KUKA KRL program: EPS_2_26115_SA7008_A_20260219035546.src

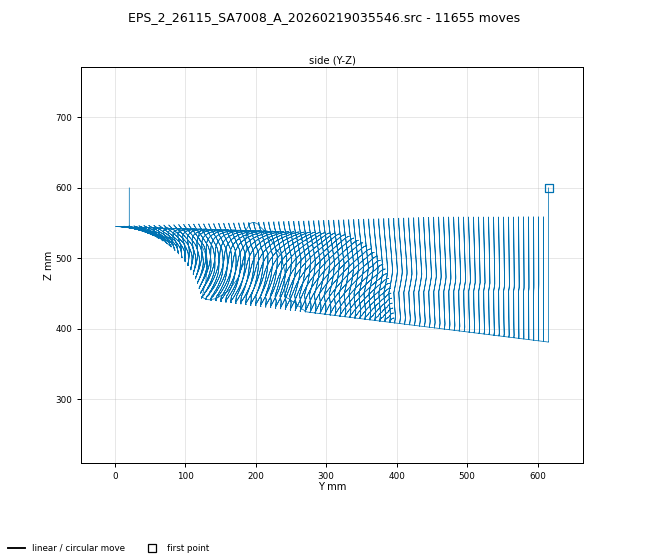
[picture p0: tool path of EPS_2_26115_SA7008_A_20260219035546.src, 11655 of 11657 moves have a stored position in this frame; points joined in program order, loops and branches not executed]
&ACCESS RVP
&REL 4
&COMMENT QRS 19112012
&PARAM EDITMASK = *
DEF PART()
EXT BAS (BAS_COMMAND :IN,REAL :IN )
INT I
BAS (#INITMOV,0 )

;KUKA QRS Post kuka4.cps  Date:22-06-2017 !

File_ID=3064

QRS_PRE_INIT()

;Init var - Until changes are made in qrs_pre_init
Outlet_Square_prg=0
Inlet_1_Square_prg=0
Inlet_2_Square_prg=0
Inlet_3_Square_prg=0
Inlet_4_Square_prg=0
Inlet_5_Square_prg=0

Outlet_1={X 0.000, Y 460.000, Z 458.500, B 0.000, E1 0.000 }
Inlet_1={X 0.000, Y 549.230, Z 433.500, B 0.000, E1 180.000 }
Outlet_1_type=201
Inlet_1_type=0
;QRS#1=Sidecore dimensions
;QRS#2=200-8" PVC SDR 35 Cut Back
;QRS#3=DeadEnd 201
;QRS#4=
;QRS#5=
;QRS#6=
;QRS#7=
;QRS#8=
;QRS#9=12-08 PSX
;QRS#10=

;QRS#11=
;QRS#12=
;QRS#13=
;QRS#14=
;QRS#15=
;QRS#16=1220x127x838 2,75'
;QRS#17=EPS Height
;QRS#18=559
;QRS#19=*
;QRS#20= UPDATED VERSION 22-06-2017
;QRS#21=*
Outlet_Square=0100
Inlet_1_Square=00
Inlet_2_Square=0
Inlet_3_Square=0
Inlet_4_Square=0
Inlet_5_Square=0
Mill_Square=1
Outlet_Square_Prg=214
Inlet_1_Square_prg=0

QRS_INIT()

$ADVANCE=5

; T1
PTP {E1 173.601,E2 173.601}
PTP {X 0,Y 615.5,A -85,B 0,C 180,E1 173.601,E2 173.601,E3 0,E4 0,E5 0,E6 0}
QRS_SPEED_INIT()
LIN {X 0,Y 615.5,Z 600,A -85,B 0,C 180,E1 173.601,E2 173.601,E3 0,E4 0,E5 0,E6 0} C_VEL
LIN {X 0,Y 615.5,Z 391.375,A -85,B 0,C 180,E1 173.601,E2 173.601} C_VEL
LIN {X 0,Y 615.5,Z 383.193,A -85,B 0,C 180,E1 173.601,E2 173.601} C_VEL
LIN {X 0,Y 615.486,Z 381.193,A -85,B 0,C 180,E1 173.415,E2 173.415} C_VEL
LIN {X 0,Y 615.489,Z 381.182,A -85,B 0,C 180,E1 170.802,E2 170.802} C_VEL
LIN {X 0,Y 615.48,Z 381.193,A -85,B 0,C 180,E1 168.139,E2 168.139} C_VEL
LIN {X 0,Y 615.481,Z 381.192,A -85,B 0,C 180,E1 165.451,E2 165.451} C_VEL
LIN {X 0,Y 615.493,Z 381.182,A -85,B 0,C 180,E1 162.73,E2 162.73} C_VEL
LIN {X 0,Y 615.49,Z 381.2,A -85,B 0,C 180,E1 159.968,E2 159.968} C_VEL
LIN {X 0,Y 615.481,Z 381.185,A -85,B 0,C 180,E1 157.156,E2 157.156} C_VEL
LIN {X 0,Y 615.481,Z 381.195,A -85,B 0,C 180,E1 154.284,E2 154.284} C_VEL
LIN {X 0,Y 615.478,Z 381.19,A -85,B 0,C 180,E1 151.55,E2 151.55} C_VEL
LIN {X 0,Y 615.485,Z 381.184,A -85,B 0,C 180,E1 148.913,E2 148.913} C_VEL
LIN {X 0,Y 615.489,Z 381.197,A -85,B 0,C 180,E1 145.979,E2 145.979} C_VEL
LIN {X 0,Y 615.485,Z 381.183,A -85,B 0,C 180,E1 143.062,E2 143.062} C_VEL
LIN {X 0,Y 615.495,Z 381.2,A -85,B 0,C 180,E1 140.251,E2 140.251} C_VEL
LIN {X 0,Y 615.477,Z 381.188,A -85,B 0,C 180,E1 137.647,E2 137.647} C_VEL
LIN {X 0,Y 615.482,Z 381.187,A -85,B 0,C 180,E1 134.932,E2 134.932} C_VEL
LIN {X 0,Y 615.481,Z 381.195,A -85,B 0,C 180,E1 132.08,E2 132.08} C_VEL
LIN {X 0,Y 615.477,Z 381.187,A -85,B 0,C 180,E1 129.75,E2 129.75} C_VEL
LIN {X 0,Y 615.477,Z 381.19,A -85,B 0,C 180,E1 126.936,E2 126.936} C_VEL
LIN {X 0,Y 615.482,Z 381.196,A -85,B 0,C 180,E1 124.701,E2 124.701} C_VEL
LIN {X 0,Y 615.49,Z 381.196,A -85,B 0,C 180,E1 122.332,E2 122.332} C_VEL
LIN {X 0,Y 615.492,Z 381.182,A -85,B 0,C 180,E1 119.405,E2 119.405} C_VEL
LIN {X 0,Y 615.486,Z 381.198,A -85,B 0,C 180,E1 116.444,E2 116.444} C_VEL
LIN {X 0,Y 615.485,Z 381.183,A -85,B 0,C 180,E1 113.556,E2 113.556} C_VEL
LIN {X 0,Y 615.488,Z 381.201,A -85,B 0,C 180,E1 110.73,E2 110.73} C_VEL
LIN {X 0,Y 615.483,Z 381.185,A -85,B 0,C 180,E1 107.957,E2 107.957} C_VEL
LIN {X 0,Y 615.478,Z 381.19,A -85,B 0,C 180,E1 105.226,E2 105.226} C_VEL
LIN {X 0,Y 615.483,Z 381.194,A -85,B 0,C 180,E1 102.53,E2 102.53} C_VEL
LIN {X 0,Y 615.498,Z 381.18,A -85,B 0,C 180,E1 99.862,E2 99.862} C_VEL
LIN {X 0,Y 615.48,Z 381.193,A -85,B 0,C 180,E1 97.215,E2 97.215} C_VEL
LIN {X 0,Y 615.48,Z 381.193,A -85,B 0,C 180,E1 94.584,E2 94.584} C_VEL
LIN {X 0,Y 615.499,Z 381.18,A -85,B 0,C 180,E1 91.963,E2 91.963} C_VEL
LIN {X 0,Y 615.48,Z 381.193,A -85,B 0,C 180,E1 89.346,E2 89.346} C_VEL
LIN {X 0,Y 615.48,Z 381.193,A -85,B 0,C 180,E1 86.727,E2 86.727} C_VEL
LIN {X 0,Y 615.498,Z 381.18,A -85,B 0,C 180,E1 84.101,E2 84.101} C_VEL
LIN {X 0,Y 615.48,Z 381.193,A -85,B 0,C 180,E1 81.463,E2 81.463} C_VEL
LIN {X 0,Y 615.48,Z 381.193,A -85,B 0,C 180,E1 78.807,E2 78.807} C_VEL
LIN {X 0,Y 615.487,Z 381.183,A -85,B 0,C 180,E1 76.065,E2 76.065} C_VEL
LIN {X 0,Y 615.489,Z 381.197,A -85,B 0,C 180,E1 73.414,E2 73.414} C_VEL
LIN {X 0,Y 615.481,Z 381.187,A -85,B 0,C 180,E1 70.662,E2 70.662} C_VEL
LIN {X 0,Y 615.478,Z 381.189,A -85,B 0,C 180,E1 67.863,E2 67.863} C_VEL
LIN {X 0,Y 615.48,Z 381.192,A -85,B 0,C 180,E1 65.008,E2 65.008} C_VEL
LIN {X 0,Y 615.479,Z 381.188,A -85,B 0,C 180,E1 62.823,E2 62.823} C_VEL
LIN {X 0,Y 615.481,Z 381.185,A -85,B 0,C 180,E1 60.205,E2 60.205} C_VEL
LIN {X 0,Y 615.493,Z 381.2,A -85,B 0,C 180,E1 57.543,E2 57.543} C_VEL
LIN {X 0,Y 615.479,Z 381.193,A -85,B 0,C 180,E1 55.185,E2 55.185} C_VEL
LIN {X 0,Y 615.485,Z 381.184,A -85,B 0,C 180,E1 52.758,E2 52.758} C_VEL
LIN {X 0,Y 615.481,Z 381.194,A -85,B 0,C 180,E1 49.911,E2 49.911} C_VEL
LIN {X 0,Y 615.5,Z 381.2,A -85,B 0,C 180,E1 47.649,E2 47.649} C_VEL
LIN {X 0,Y 615.481,Z 381.185,A -85,B 0,C 180,E1 44.932,E2 44.932} C_VEL
LIN {X 0,Y 615.482,Z 381.193,A -85,B 0,C 180,E1 42.08,E2 42.08} C_VEL
LIN {X 0,Y 615.495,Z 381.2,A -85,B 0,C 180,E1 39.749,E2 39.749} C_VEL
LIN {X 0,Y 615.485,Z 381.183,A -85,B 0,C 180,E1 36.937,E2 36.937} C_VEL
LIN {X 0,Y 615.488,Z 381.197,A -85,B 0,C 180,E1 34.021,E2 34.021} C_VEL
LIN {X 0,Y 615.483,Z 381.184,A -85,B 0,C 180,E1 31.086,E2 31.086} C_VEL
LIN {X 0,Y 615.478,Z 381.19,A -85,B 0,C 180,E1 28.45,E2 28.45} C_VEL
LIN {X 0,Y 615.484,Z 381.194,A -85,B 0,C 180,E1 25.715,E2 25.715} C_VEL
LIN {X 0,Y 615.481,Z 381.185,A -85,B 0,C 180,E1 22.844,E2 22.844} C_VEL
LIN {X 0,Y 615.492,Z 381.2,A -85,B 0,C 180,E1 20.032,E2 20.032} C_VEL
LIN {X 0,Y 615.491,Z 381.182,A -85,B 0,C 180,E1 17.27,E2 17.27} C_VEL
LIN {X 0,Y 615.481,Z 381.192,A -85,B 0,C 180,E1 14.549,E2 14.549} C_VEL
LIN {X 0,Y 615.483,Z 381.192,A -85,B 0,C 180,E1 11.86,E2 11.86} C_VEL
LIN {X 0,Y 615.489,Z 381.182,A -85,B 0,C 180,E1 9.198,E2 9.198} C_VEL
LIN {X 0,Y 615.487,Z 381.193,A -85,B 0,C 180,E1 6.556,E2 6.556} C_VEL
LIN {X 0,Y 615.482,Z 381.191,A -85,B 0,C 180,E1 3.928,E2 3.928} C_VEL
LIN {X 0,Y 615.487,Z 381.183,A -85,B 0,C 180,E1 1.308,E2 1.308} C_VEL
LIN {X 0,Y 615.487,Z 381.193,A -85,B 0,C 180,E1 -1.309,E2 -1.309} C_VEL
LIN {X 0,Y 615.483,Z 381.191,A -85,B 0,C 180,E1 -3.929,E2 -3.929} C_VEL
LIN {X 0,Y 615.486,Z 381.183,A -85,B 0,C 180,E1 -6.583,E2 -6.583} C_VEL
LIN {X 0,Y 615.489,Z 381.193,A -85,B 0,C 180,E1 -9.199,E2 -9.199} C_VEL
LIN {X 0,Y 615.483,Z 381.19,A -85,B 0,C 180,E1 -11.861,E2 -11.861} C_VEL
LIN {X 0,Y 615.481,Z 381.184,A -85,B 0,C 180,E1 -14.55,E2 -14.55} C_VEL
LIN {X 0,Y 615.494,Z 381.199,A -85,B 0,C 180,E1 -17.271,E2 -17.271} C_VEL
LIN {X 0,Y 615.491,Z 381.183,A -85,B 0,C 180,E1 -20.033,E2 -20.033} C_VEL
LIN {X 0,Y 615.481,Z 381.191,A -85,B 0,C 180,E1 -22.845,E2 -22.845} C_VEL
LIN {X 0,Y 615.484,Z 381.188,A -85,B 0,C 180,E1 -25.716,E2 -25.716} C_VEL
LIN {X 0,Y 615.478,Z 381.186,A -85,B 0,C 180,E1 -28.45,E2 -28.45} C_VEL
LIN {X 0,Y 615.49,Z 381.201,A -85,B 0,C 180,E1 -31.088,E2 -31.088} C_VEL
LIN {X 0,Y 615.489,Z 381.182,A -85,B 0,C 180,E1 -34.022,E2 -34.022} C_VEL
LIN {X 0,Y 615.493,Z 381.198,A -85,B 0,C 180,E1 -36.938,E2 -36.938} C_VEL
LIN {X 0,Y 615.492,Z 381.183,A -85,B 0,C 180,E1 -39.75,E2 -39.75} C_VEL
LIN {X 0,Y 615.477,Z 381.188,A -85,B 0,C 180,E1 -42.354,E2 -42.354} C_VEL
LIN {X 0,Y 615.491,Z 381.196,A -85,B 0,C 180,E1 -45.069,E2 -45.069} C_VEL
LIN {X 0,Y 615.485,Z 381.183,A -85,B 0,C 180,E1 -47.921,E2 -47.921} C_VEL
LIN {X 0,Y 615.499,Z 381.333,A -85,B 0,C 180,E1 -48.717,E2 -48.717} C_VEL
LIN {X 0,Y 615.485,Z 386.318,A -85,B 0,C 180,E1 -51.096,E2 -51.096} C_VEL
LIN {X 0,Y 615.486,Z 391.692,A -85,B 0,C 180,E1 -53.576,E2 -53.576} C_VEL
LIN {X 0,Y 615.491,Z 398.17,A -85,B 0,C 180,E1 -56.466,E2 -56.466} C_VEL
LIN {X 0,Y 615.478,Z 404.223,A -85,B 0,C 180,E1 -59.08,E2 -59.08} C_VEL
LIN {X 0,Y 615.495,Z 410.088,A -85,B 0,C 180,E1 -61.549,E2 -61.549} C_VEL
LIN {X 0,Y 615.498,Z 417.097,A -85,B 0,C 180,E1 -64.43,E2 -64.43} C_VEL
LIN {X 0,Y 615.483,Z 423.897,A -85,B 0,C 180,E1 -67.155,E2 -67.155} C_VEL
LIN {X 0,Y 615.479,Z 431.039,A -85,B 0,C 180,E1 -69.967,E2 -69.967} C_VEL
LIN {X 0,Y 615.479,Z 438.188,A -85,B 0,C 180,E1 -72.729,E2 -72.729} C_VEL
LIN {X 0,Y 615.483,Z 445.321,A -85,B 0,C 180,E1 -75.451,E2 -75.451} C_VEL
LIN {X 0,Y 615.486,Z 452.468,A -85,B 0,C 180,E1 -78.139,E2 -78.139} C_VEL
LIN {X 0,Y 615.491,Z 453.075,A -85,B 0,C 180,E1 -78.369,E2 -78.369} C_VEL
LIN {X 0,Y 615.493,Z 468.86,A -85,B 0,C 180,E1 -78.724,E2 -78.724} C_VEL
LIN {X 0,Y 615.492,Z 481.787,A -85,B 0,C 180,E1 -79.157,E2 -79.157} C_VEL
LIN {X 0,Y 615.478,Z 494.043,A -85,B 0,C 180,E1 -79.722,E2 -79.722} C_VEL
LIN {X 0,Y 615.498,Z 505.266,A -85,B 0,C 180,E1 -80.387,E2 -80.387} C_VEL
LIN {X 0,Y 615.498,Z 515.389,A -85,B 0,C 180,E1 -81.133,E2 -81.133} C_VEL
LIN {X 0,Y 615.498,Z 524.474,A -85,B 0,C 180,E1 -81.959,E2 -81.959} C_VEL
LIN {X 0,Y 615.498,Z 533.261,A -85,B 0,C 180,E1 -82.943,E2 -82.943} C_VEL
LIN {X 0,Y 615.496,Z 540.416,A -85,B 0,C 180,E1 -83.937,E2 -83.937} C_VEL
LIN {X 0,Y 615.496,Z 546.872,A -85,B 0,C 180,E1 -85.087,E2 -85.087} C_VEL
LIN {X 0,Y 615.496,Z 551.141,A -85,B 0,C 180,E1 -86.071,E2 -86.071} C_VEL
LIN {X 0,Y 615.495,Z 553.398,A -85,B 0,C 180,E1 -86.727,E2 -86.727} C_VEL
LIN {X 0,Y 615.497,Z 555.233,A -85,B 0,C 180,E1 -87.382,E2 -87.382} C_VEL
LIN {X 0,Y 615.499,Z 556.607,A -85,B 0,C 180,E1 -88.037,E2 -88.037} C_VEL
LIN {X 0,Y 615.496,Z 558.173,A -85,B 0,C 180,E1 -89.346,E2 -89.346} C_VEL
LIN {X 0,Y 615.494,Z 558.389,A -85,B 0,C 180,E1 -90,E2 -90} C_VEL
LIN {X 0,Y 615.496,Z 557.58,A -85,B 0,C 180,E1 -91.308,E2 -91.308} C_VEL
LIN {X 0,Y 615.499,Z 556.608,A -85,B 0,C 180,E1 -91.963,E2 -91.963} C_VEL
LIN {X 0,Y 615.497,Z 555.233,A -85,B 0,C 180,E1 -92.618,E2 -92.618} C_VEL
LIN {X 0,Y 615.496,Z 552.35,A -85,B 0,C 180,E1 -93.6,E2 -93.6} C_VEL
LIN {X 0,Y 615.498,Z 548.442,A -85,B 0,C 180,E1 -94.584,E2 -94.584} C_VEL
LIN {X 0,Y 615.499,Z 543.406,A -85,B 0,C 180,E1 -95.569,E2 -95.569} C_VEL
LIN {X 0,Y 615.497,Z 536.87,A -85,B 0,C 180,E1 -96.583,E2 -96.583} C_VEL
LIN {X 0,Y 615.497,Z 529.135,A -85,B 0,C 180,E1 -97.545,E2 -97.545} C_VEL
LIN {X 0,Y 615.498,Z 521.048,A -85,B 0,C 180,E1 -98.371,E2 -98.371} C_VEL
LIN {X 0,Y 615.499,Z 511.171,A -85,B 0,C 180,E1 -99.198,E2 -99.198} C_VEL
LIN {X 0,Y 615.491,Z 499.986,A -85,B 0,C 180,E1 -99.945,E2 -99.945} C_VEL
LIN {X 0,Y 615.481,Z 489.03,A -85,B 0,C 180,E1 -100.527,E2 -100.527} C_VEL
LIN {X 0,Y 615.488,Z 476.477,A -85,B 0,C 180,E1 -101.04,E2 -101.04} C_VEL
LIN {X 0,Y 615.497,Z 464.077,A -85,B 0,C 180,E1 -101.401,E2 -101.401} C_VEL
LIN {X 0,Y 615.491,Z 453.076,A -85,B 0,C 180,E1 -101.631,E2 -101.631} C_VEL
LIN {X 0,Y 615.487,Z 446.962,A -85,B 0,C 180,E1 -103.932,E2 -103.932} C_VEL
LIN {X 0,Y 615.489,Z 439.966,A -85,B 0,C 180,E1 -106.586,E2 -106.586} C_VEL
LIN {X 0,Y 615.481,Z 432.836,A -85,B 0,C 180,E1 -109.338,E2 -109.338} C_VEL
LIN {X 0,Y 615.478,Z 425.679,A -85,B 0,C 180,E1 -112.136,E2 -112.136} C_VEL
LIN {X 0,Y 615.478,Z 418.538,A -85,B 0,C 180,E1 -114.992,E2 -114.992} C_VEL
LIN {X 0,Y 615.478,Z 413.169,A -85,B 0,C 180,E1 -117.177,E2 -117.177} C_VEL
LIN {X 0,Y 615.486,Z 406.877,A -85,B 0,C 180,E1 -119.794,E2 -119.794} C_VEL
LIN {X 0,Y 615.494,Z 400.647,A -85,B 0,C 180,E1 -122.456,E2 -122.456} C_VEL
LIN {X 0,Y 615.479,Z 395.273,A -85,B 0,C 180,E1 -124.815,E2 -124.815} C_VEL
LIN {X 0,Y 615.487,Z 389.901,A -85,B 0,C 180,E1 -127.241,E2 -127.241} C_VEL
LIN {X 0,Y 615.481,Z 383.818,A -85,B 0,C 180,E1 -130.088,E2 -130.088} C_VEL
LIN {X 0,Y 615.494,Z 381.193,A -85,B 0,C 180,E1 -131.378,E2 -131.378} C_VEL
LIN {X 0,Y 615.491,Z 381.182,A -85,B 0,C 180,E1 -134.148,E2 -134.148} C_VEL
LIN {X 0,Y 615.492,Z 381.198,A -85,B 0,C 180,E1 -136.951,E2 -136.951} C_VEL
LIN {X 0,Y 615.481,Z 381.192,A -85,B 0,C 180,E1 -139.393,E2 -139.393} C_VEL
LIN {X 0,Y 615.483,Z 381.183,A -85,B 0,C 180,E1 -141.987,E2 -141.987} C_VEL
LIN {X 0,Y 615.485,Z 381.187,A -85,B 0,C 180,E1 -144.384,E2 -144.384} C_VEL
LIN {X 0,Y 615.484,Z 381.198,A -85,B 0,C 180,E1 -146.763,E2 -146.763} C_VEL
LIN {X 0,Y 615.489,Z 381.195,A -85,B 0,C 180,E1 -149.08,E2 -149.08} C_VEL
LIN {X 0,Y 615.478,Z 381.186,A -85,B 0,C 180,E1 -151.55,E2 -151.55} C_VEL
LIN {X 0,Y 615.484,Z 381.188,A -85,B 0,C 180,E1 -154.284,E2 -154.284} C_VEL
LIN {X 0,Y 615.481,Z 381.191,A -85,B 0,C 180,E1 -157.155,E2 -157.155} C_VEL
LIN {X 0,Y 615.491,Z 381.183,A -85,B 0,C 180,E1 -159.967,E2 -159.967} C_VEL
LIN {X 0,Y 615.494,Z 381.199,A -85,B 0,C 180,E1 -162.729,E2 -162.729} C_VEL
LIN {X 0,Y 615.481,Z 381.184,A -85,B 0,C 180,E1 -165.45,E2 -165.45} C_VEL
LIN {X 0,Y 615.483,Z 381.19,A -85,B 0,C 180,E1 -168.139,E2 -168.139} C_VEL
LIN {X 0,Y 615.489,Z 381.193,A -85,B 0,C 180,E1 -170.801,E2 -170.801} C_VEL
LIN {X 0,Y 615.487,Z 381.182,A -85,B 0,C 180,E1 -173.443,E2 -173.443} C_VEL
LIN {X 0,Y 615.483,Z 381.191,A -85,B 0,C 180,E1 -176.071,E2 -176.071} C_VEL
LIN {X 0,Y 615.487,Z 381.193,A -85,B 0,C 180,E1 -178.691,E2 -178.691} C_VEL
LIN {X 0,Y 615.487,Z 381.183,A -85,B 0,C 180,E1 -181.308,E2 -181.308} C_VEL
LIN {X 0,Y 615.48,Z 381.192,A -85,B 0,C 180,E1 -183.928,E2 -183.928} C_VEL
LIN {X 0,Y 615.486,Z 381.193,A -85,B 0,C 180,E1 -186.585,E2 -186.585} C_VEL
LIN {X 0,Y 614.81,Z 381.332,A -85,B 0,C 180,E1 -187.131,E2 -187.131} C_VEL
LIN {X 0,Y 611.977,Z 381.755,A -85,B 0,C 180,E1 -188.017,E2 -188.017} C_VEL
LIN {X 0,Y 609.586,Z 382.06,A -85,B 0,C 180,E1 -188.729,E2 -188.729} C_VEL
LIN {X 0,Y 608.549,Z 382.177,A -85,B 0,C 180,E1 -189.279,E2 -189.279} C_VEL
LIN {X 0,Y 608.459,Z 382.187,A -85,B 0,C 180,E1 -189.465,E2 -189.465} C_VEL
LIN {X 0,Y 608.456,Z 382.194,A -85,B 0,C 180,E1 -191.999,E2 -191.999} C_VEL
LIN {X 0,Y 608.471,Z 382.187,A -85,B 0,C 180,E1 -194.72,E2 -194.72} C_VEL
LIN {X 0,Y 608.457,Z 382.188,A -85,B 0,C 180,E1 -197.476,E2 -197.476} C_VEL
LIN {X 0,Y 608.46,Z 382.194,A -85,B 0,C 180,E1 -200.274,E2 -200.274} C_VEL
LIN {X 0,Y 608.449,Z 382.191,A -85,B 0,C 180,E1 -202.476,E2 -202.476} C_VEL
LIN {X 0,Y 608.455,Z 382.189,A -85,B 0,C 180,E1 -204.571,E2 -204.571} C_VEL
LIN {X 0,Y 608.483,Z 382.184,A -85,B 0,C 180,E1 -207.21,E2 -207.21} C_VEL
LIN {X 0,Y 608.47,Z 382.195,A -85,B 0,C 180,E1 -209.974,E2 -209.974} C_VEL
LIN {X 0,Y 608.452,Z 382.189,A -85,B 0,C 180,E1 -212.523,E2 -212.523} C_VEL
LIN {X 0,Y 608.442,Z 382.191,A -85,B 0,C 180,E1 -215.277,E2 -215.277} C_VEL
LIN {X 0,Y 608.465,Z 382.196,A -85,B 0,C 180,E1 -217.746,E2 -217.746} C_VEL
LIN {X 0,Y 608.448,Z 382.19,A -85,B 0,C 180,E1 -220.33,E2 -220.33} C_VEL
LIN {X 0,Y 608.449,Z 382.188,A -85,B 0,C 180,E1 -222.96,E2 -222.96} C_VEL
LIN {X 0,Y 608.458,Z 382.197,A -85,B 0,C 180,E1 -225.735,E2 -225.735} C_VEL
LIN {X 0,Y 608.462,Z 382.186,A -85,B 0,C 180,E1 -228.657,E2 -228.657} C_VEL
LIN {X 0,Y 608.463,Z 382.193,A -85,B 0,C 180,E1 -231.412,E2 -231.412} C_VEL
LIN {X 0,Y 608.471,Z 382.189,A -85,B 0,C 180,E1 -233.951,E2 -233.951} C_VEL
LIN {X 0,Y 608.465,Z 382.186,A -85,B 0,C 180,E1 -236.33,E2 -236.33} C_VEL
LIN {X 0,Y 608.472,Z 382.186,A -85,B 0,C 180,E1 -238.728,E2 -238.728} C_VEL
LIN {X 0,Y 608.473,Z 382.195,A -85,B 0,C 180,E1 -241.379,E2 -241.379} C_VEL
LIN {X 0,Y 608.474,Z 382.185,A -85,B 0,C 180,E1 -244.278,E2 -244.278} C_VEL
LIN {X 0,Y 608.448,Z 382.191,A -85,B 0,C 180,E1 -246.876,E2 -246.876} C_VEL
LIN {X 0,Y 608.459,Z 382.19,A -85,B 0,C 180,E1 -249.726,E2 -249.726} C_VEL
LIN {X 0,Y 608.447,Z 382.189,A -85,B 0,C 180,E1 -252.524,E2 -252.524} C_VEL
LIN {X 0,Y 608.471,Z 382.195,A -85,B 0,C 180,E1 -255.28,E2 -255.28} C_VEL
LIN {X 0,Y 608.461,Z 382.187,A -85,B 0,C 180,E1 -258.001,E2 -258.001} C_VEL
LIN {X 0,Y 608.467,Z 382.189,A -85,B 0,C 180,E1 -260.694,E2 -260.694} C_VEL
LIN {X 0,Y 608.474,Z 382.191,A -85,B 0,C 180,E1 -263.368,E2 -263.368} C_VEL
LIN {X 0,Y 608.455,Z 382.187,A -85,B 0,C 180,E1 -266.026,E2 -266.026} C_VEL
LIN {X 0,Y 608.465,Z 382.191,A -85,B 0,C 180,E1 -268.676,E2 -268.676} C_VEL
LIN {X 0,Y 608.465,Z 382.191,A -85,B 0,C 180,E1 -271.324,E2 -271.324} C_VEL
LIN {X 0,Y 608.455,Z 382.187,A -85,B 0,C 180,E1 -273.974,E2 -273.974} C_VEL
LIN {X 0,Y 608.475,Z 382.191,A -85,B 0,C 180,E1 -276.633,E2 -276.633} C_VEL
LIN {X 0,Y 608.467,Z 382.189,A -85,B 0,C 180,E1 -279.306,E2 -279.306} C_VEL
LIN {X 0,Y 608.461,Z 382.187,A -85,B 0,C 180,E1 -282,E2 -282} C_VEL
LIN {X 0,Y 608.471,Z 382.195,A -85,B 0,C 180,E1 -284.721,E2 -284.721} C_VEL
LIN {X 0,Y 608.447,Z 382.189,A -85,B 0,C 180,E1 -287.477,E2 -287.477} C_VEL
LIN {X 0,Y 608.459,Z 382.19,A -85,B 0,C 180,E1 -290.274,E2 -290.274} C_VEL
LIN {X 0,Y 608.45,Z 382.191,A -85,B 0,C 180,E1 -293.124,E2 -293.124} C_VEL
LIN {X 0,Y 608.474,Z 382.185,A -85,B 0,C 180,E1 -295.722,E2 -295.722} C_VEL
LIN {X 0,Y 608.474,Z 382.194,A -85,B 0,C 180,E1 -298.621,E2 -298.621} C_VEL
LIN {X 0,Y 608.472,Z 382.185,A -85,B 0,C 180,E1 -301.316,E2 -301.316} C_VEL
LIN {X 0,Y 608.473,Z 382.185,A -85,B 0,C 180,E1 -303.736,E2 -303.736} C_VEL
LIN {X 0,Y 608.472,Z 382.19,A -85,B 0,C 180,E1 -306.09,E2 -306.09} C_VEL
LIN {X 0,Y 608.464,Z 382.193,A -85,B 0,C 180,E1 -308.588,E2 -308.588} C_VEL
LIN {X 0,Y 608.462,Z 382.186,A -85,B 0,C 180,E1 -311.343,E2 -311.343} C_VEL
LIN {X 0,Y 608.458,Z 382.197,A -85,B 0,C 180,E1 -314.265,E2 -314.265} C_VEL
LIN {X 0,Y 608.449,Z 382.188,A -85,B 0,C 180,E1 -317.04,E2 -317.04} C_VEL
LIN {X 0,Y 608.447,Z 382.19,A -85,B 0,C 180,E1 -319.697,E2 -319.697} C_VEL
LIN {X 0,Y 608.466,Z 382.196,A -85,B 0,C 180,E1 -322.254,E2 -322.254} C_VEL
LIN {X 0,Y 608.48,Z 382.184,A -85,B 0,C 180,E1 -325.09,E2 -325.09} C_VEL
LIN {X 0,Y 608.46,Z 382.194,A -85,B 0,C 180,E1 -327.906,E2 -327.906} C_VEL
LIN {X 0,Y 608.475,Z 382.193,A -85,B 0,C 180,E1 -330.221,E2 -330.221} C_VEL
LIN {X 0,Y 608.451,Z 382.188,A -85,B 0,C 180,E1 -333.226,E2 -333.226} C_VEL
LIN {X 0,Y 608.467,Z 382.193,A -85,B 0,C 180,E1 -336.156,E2 -336.156} C_VEL
LIN {X 0,Y 608.468,Z 382.19,A -85,B 0,C 180,E1 -338.309,E2 -338.309} C_VEL
LIN {X 0,Y 608.45,Z 382.188,A -85,B 0,C 180,E1 -341.131,E2 -341.131} C_VEL
LIN {X 0,Y 608.46,Z 382.197,A -85,B 0,C 180,E1 -343.907,E2 -343.907} C_VEL
LIN {X 0,Y 608.468,Z 382.186,A -85,B 0,C 180,E1 -346.644,E2 -346.644} C_VEL
LIN {X 0,Y 608.461,Z 382.19,A -85,B 0,C 180,E1 -349.351,E2 -349.351} C_VEL
LIN {X 0,Y 608.473,Z 382.19,A -85,B 0,C 180,E1 -352.033,E2 -352.033} C_VEL
LIN {X 0,Y 608.466,Z 382.186,A -85,B 0,C 180,E1 -354.699,E2 -354.699} C_VEL
LIN {X 0,Y 608.478,Z 382.19,A -85,B 0,C 180,E1 -357.352,E2 -357.352} C_VEL
LIN {X 0,Y 608.473,Z 382.189,A -85,B 0,C 180,E1 -360,E2 -360} C_VEL
LIN {X 0,Y 608.478,Z 382.184,A -85,B 0,C 180,E1 -362.648,E2 -362.648} C_VEL
LIN {X 0,Y 608.466,Z 382.192,A -85,B 0,C 180,E1 -365.302,E2 -365.302} C_VEL
LIN {X 0,Y 608.475,Z 382.188,A -85,B 0,C 180,E1 -367.967,E2 -367.967} C_VEL
LIN {X 0,Y 608.461,Z 382.187,A -85,B 0,C 180,E1 -370.65,E2 -370.65} C_VEL
LIN {X 0,Y 608.468,Z 382.195,A -85,B 0,C 180,E1 -373.357,E2 -373.357} C_VEL
LIN {X 0,Y 608.457,Z 382.188,A -85,B 0,C 180,E1 -376.094,E2 -376.094} C_VEL
LIN {X 0,Y 608.452,Z 382.191,A -85,B 0,C 180,E1 -378.87,E2 -378.87} C_VEL
LIN {X 0,Y 608.473,Z 382.189,A -85,B 0,C 180,E1 -381.692,E2 -381.692} C_VEL
LIN {X 0,Y 608.456,Z 382.188,A -85,B 0,C 180,E1 -384.571,E2 -384.571} C_VEL
LIN {X 0,Y 608.485,Z 382.194,A -85,B 0,C 180,E1 -387.21,E2 -387.21} C_VEL
LIN {X 0,Y 608.469,Z 382.186,A -85,B 0,C 180,E1 -389.973,E2 -389.973} C_VEL
LIN {X 0,Y 608.453,Z 382.189,A -85,B 0,C 180,E1 -392.522,E2 -392.522} C_VEL
LIN {X 0,Y 608.445,Z 382.195,A -85,B 0,C 180,E1 -395.278,E2 -395.278} C_VEL
LIN {X 0,Y 608.469,Z 382.186,A -85,B 0,C 180,E1 -397.747,E2 -397.747} C_VEL
LIN {X 0,Y 608.448,Z 382.189,A -85,B 0,C 180,E1 -400.329,E2 -400.329} C_VEL
LIN {X 0,Y 608.473,Z 382.19,A -85,B 0,C 180,E1 -403.31,E2 -403.31} C_VEL
LIN {X 0,Y 608.469,Z 382.186,A -85,B 0,C 180,E1 -406.131,E2 -406.131} C_VEL
LIN {X 0,Y 608.48,Z 382.305,A -85,B 0,C 180,E1 -408.522,E2 -408.522} C_VEL
LIN {X 0,Y 608.476,Z 386.675,A -85,B 0,C 180,E1 -410.702,E2 -410.702} C_VEL
LIN {X 0,Y 608.469,Z 391.768,A -85,B 0,C 180,E1 -413.086,E2 -413.086} C_VEL
LIN {X 0,Y 608.467,Z 397.158,A -85,B 0,C 180,E1 -415.531,E2 -415.531} C_VEL
LIN {X 0,Y 608.474,Z 402.547,A -85,B 0,C 180,E1 -417.906,E2 -417.906} C_VEL
LIN {X 0,Y 608.472,Z 407.937,A -85,B 0,C 180,E1 -420.221,E2 -420.221} C_VEL
LIN {X 0,Y 608.453,Z 414.087,A -85,B 0,C 180,E1 -422.798,E2 -422.798} C_VEL
LIN {X 0,Y 608.452,Z 420.513,A -85,B 0,C 180,E1 -425.429,E2 -425.429} C_VEL
LIN {X 0,Y 608.441,Z 427.699,A -85,B 0,C 180,E1 -428.308,E2 -428.308} C_VEL
LIN {X 0,Y 608.454,Z 435.294,A -85,B 0,C 180,E1 -431.29,E2 -431.29} C_VEL
LIN {X 0,Y 608.442,Z 442.071,A -85,B 0,C 180,E1 -433.906,E2 -433.906} C_VEL
LIN {X 0,Y 608.439,Z 449.257,A -85,B 0,C 180,E1 -436.643,E2 -436.643} C_VEL
LIN {X 0,Y 608.457,Z 453.617,A -85,B 0,C 180,E1 -438.254,E2 -438.254} C_VEL
LIN {X 0,Y 608.543,Z 466.701,A -85,B 0,C 180,E1 -438.53,E2 -438.53} C_VEL
LIN {X 0,Y 608.515,Z 480.159,A -85,B 0,C 180,E1 -438.964,E2 -438.964} C_VEL
LIN {X 0,Y 608.499,Z 492.63,A -85,B 0,C 180,E1 -439.519,E2 -439.519} C_VEL
LIN {X 0,Y 608.488,Z 504.197,A -85,B 0,C 180,E1 -440.191,E2 -440.191} C_VEL
LIN {X 0,Y 608.485,Z 514.594,A -85,B 0,C 180,E1 -440.946,E2 -440.946} C_VEL
LIN {X 0,Y 608.475,Z 523.112,A -85,B 0,C 180,E1 -441.699,E2 -441.699} C_VEL
LIN {X 0,Y 608.471,Z 530.959,A -85,B 0,C 180,E1 -442.534,E2 -442.534} C_VEL
LIN {X 0,Y 608.461,Z 538.286,A -85,B 0,C 180,E1 -443.485,E2 -443.485} C_VEL
LIN {X 0,Y 608.45,Z 543.865,A -85,B 0,C 180,E1 -444.366,E2 -444.366} C_VEL
LIN {X 0,Y 608.432,Z 548.95,A -85,B 0,C 180,E1 -445.362,E2 -445.362} C_VEL
LIN {X 0,Y 608.449,Z 552.896,A -85,B 0,C 180,E1 -446.358,E2 -446.358} C_VEL
LIN {X 0,Y 608.425,Z 555.808,A -85,B 0,C 180,E1 -447.352,E2 -447.352} C_VEL
LIN {X 0,Y 608.444,Z 557.201,A -85,B 0,C 180,E1 -448.014,E2 -448.014} C_VEL
LIN {X 0,Y 608.438,Z 558.783,A -85,B 0,C 180,E1 -449.338,E2 -449.338} C_VEL
LIN {X 0,Y 608.434,Z 558.999,A -85,B 0,C 180,E1 -450,E2 -450} C_VEL
LIN {X 0,Y 608.448,Z 558.184,A -85,B 0,C 180,E1 -451.324,E2 -451.324} C_VEL
LIN {X 0,Y 608.444,Z 557.201,A -85,B 0,C 180,E1 -451.986,E2 -451.986} C_VEL
LIN {X 0,Y 608.425,Z 555.809,A -85,B 0,C 180,E1 -452.648,E2 -452.648} C_VEL
LIN {X 0,Y 608.449,Z 552.897,A -85,B 0,C 180,E1 -453.642,E2 -453.642} C_VEL
LIN {X 0,Y 608.432,Z 548.951,A -85,B 0,C 180,E1 -454.638,E2 -454.638} C_VEL
LIN {X 0,Y 608.437,Z 542.878,A -85,B 0,C 180,E1 -455.801,E2 -455.801} C_VEL
LIN {X 0,Y 608.462,Z 536.237,A -85,B 0,C 180,E1 -456.799,E2 -456.799} C_VEL
LIN {X 0,Y 608.455,Z 527.992,A -85,B 0,C 180,E1 -457.8,E2 -457.8} C_VEL
LIN {X 0,Y 608.472,Z 519.536,A -85,B 0,C 180,E1 -458.636,E2 -458.636} C_VEL
LIN {X 0,Y 608.481,Z 509.093,A -85,B 0,C 180,E1 -459.473,E2 -459.473} C_VEL
LIN {X 0,Y 608.491,Z 498.76,A -85,B 0,C 180,E1 -460.144,E2 -460.144} C_VEL
LIN {X 0,Y 608.517,Z 487.265,A -85,B 0,C 180,E1 -460.74,E2 -460.74} C_VEL
LIN {X 0,Y 608.536,Z 474.893,A -85,B 0,C 180,E1 -461.224,E2 -461.224} C_VEL
LIN {X 0,Y 608.546,Z 461.449,A -85,B 0,C 180,E1 -461.596,E2 -461.596} C_VEL
LIN {X 0,Y 608.436,Z 453.468,A -85,B 0,C 180,E1 -461.767,E2 -461.767} C_VEL
LIN {X 0,Y 608.431,Z 447.461,A -85,B 0,C 180,E1 -464.038,E2 -464.038} C_VEL
LIN {X 0,Y 608.446,Z 440.275,A -85,B 0,C 180,E1 -466.784,E2 -466.784} C_VEL
LIN {X 0,Y 608.447,Z 433.089,A -85,B 0,C 180,E1 -469.57,E2 -469.57} C_VEL
LIN {X 0,Y 608.441,Z 427.699,A -85,B 0,C 180,E1 -471.692,E2 -471.692} C_VEL
LIN {X 0,Y 608.452,Z 420.513,A -85,B 0,C 180,E1 -474.571,E2 -474.571} C_VEL
LIN {X 0,Y 608.452,Z 414.088,A -85,B 0,C 180,E1 -477.202,E2 -477.202} C_VEL
LIN {X 0,Y 608.47,Z 407.485,A -85,B 0,C 180,E1 -479.971,E2 -479.971} C_VEL
LIN {X 0,Y 608.493,Z 401.552,A -85,B 0,C 180,E1 -482.526,E2 -482.526} C_VEL
LIN {X 0,Y 608.476,Z 395.362,A -85,B 0,C 180,E1 -485.275,E2 -485.275} C_VEL
LIN {X 0,Y 608.49,Z 388.906,A -85,B 0,C 180,E1 -488.243,E2 -488.243} C_VEL
LIN {X 0,Y 608.539,Z 382.52,A -85,B 0,C 180,E1 -491.35,E2 -491.35} C_VEL
LIN {X 0,Y 608.461,Z 382.189,A -85,B 0,C 180,E1 -492.06,E2 -492.06} C_VEL
LIN {X 0,Y 608.458,Z 382.193,A -85,B 0,C 180,E1 -494.795,E2 -494.795} C_VEL
LIN {X 0,Y 608.457,Z 382.198,A -85,B 0,C 180,E1 -497.04,E2 -497.04} C_VEL
LIN {X 0,Y 608.448,Z 382.189,A -85,B 0,C 180,E1 -499.696,E2 -499.696} C_VEL
LIN {X 0,Y 608.468,Z 382.186,A -85,B 0,C 180,E1 -502.253,E2 -502.253} C_VEL
LIN {X 0,Y 608.481,Z 382.192,A -85,B 0,C 180,E1 -505.089,E2 -505.089} C_VEL
LIN {X 0,Y 608.46,Z 382.186,A -85,B 0,C 180,E1 -507.905,E2 -507.905} C_VEL
LIN {X 0,Y 608.472,Z 382.186,A -85,B 0,C 180,E1 -510.22,E2 -510.22} C_VEL
LIN {X 0,Y 608.483,Z 382.194,A -85,B 0,C 180,E1 -512.79,E2 -512.79} C_VEL
LIN {X 0,Y 608.455,Z 382.188,A -85,B 0,C 180,E1 -515.429,E2 -515.429} C_VEL
LIN {X 0,Y 608.473,Z 382.189,A -85,B 0,C 180,E1 -518.308,E2 -518.308} C_VEL
LIN {X 0,Y 608.463,Z 382.188,A -85,B 0,C 180,E1 -521.283,E2 -521.283} C_VEL
LIN {X 0,Y 608.457,Z 382.188,A -85,B 0,C 180,E1 -523.906,E2 -523.906} C_VEL
LIN {X 0,Y 608.468,Z 382.196,A -85,B 0,C 180,E1 -526.643,E2 -526.643} C_VEL
LIN {X 0,Y 608.461,Z 382.187,A -85,B 0,C 180,E1 -529.35,E2 -529.35} C_VEL
LIN {X 0,Y 608.474,Z 382.188,A -85,B 0,C 180,E1 -532.033,E2 -532.033} C_VEL
LIN {X 0,Y 608.466,Z 382.192,A -85,B 0,C 180,E1 -534.698,E2 -534.698} C_VEL
LIN {X 0,Y 608.478,Z 382.184,A -85,B 0,C 180,E1 -537.352,E2 -537.352} C_VEL
LIN {X 0,Y 608.471,Z 382.189,A -85,B 0,C 180,E1 -540,E2 -540} C_VEL
LIN {X 0,Y 608.478,Z 382.19,A -85,B 0,C 180,E1 -542.648,E2 -542.648} C_VEL
LIN {X 0,Y 608.466,Z 382.186,A -85,B 0,C 180,E1 -545.301,E2 -545.301} C_VEL
LIN {X 0,Y 608.472,Z 382.19,A -85,B 0,C 180,E1 -547.967,E2 -547.967} C_VEL
LIN {X 0,Y 608.459,Z 382.187,A -85,B 0,C 180,E1 -549.465,E2 -549.465} C_VEL
LIN {X 0,Y 607.776,Z 382.28,A -85,B 0,C 180,E1 -550.018,E2 -550.018} C_VEL
LIN {X 0,Y 604.918,Z 382.639,A -85,B 0,C 180,E1 -550.915,E2 -550.915} C_VEL
LIN {X 0,Y 602.516,Z 382.939,A -85,B 0,C 180,E1 -551.636,E2 -551.636} C_VEL
LIN {X 0,Y 601.488,Z 383.066,A -85,B 0,C 180,E1 -552.193,E2 -552.193} C_VEL
LIN {X 0,Y 601.406,Z 383.071,A -85,B 0,C 180,E1 -552.381,E2 -552.381} C_VEL
LIN {X 0,Y 601.426,Z 383.063,A -85,B 0,C 180,E1 -554.897,E2 -554.897} C_VEL
LIN {X 0,Y 601.429,Z 383.063,A -85,B 0,C 180,E1 -556.986,E2 -556.986} C_VEL
LIN {X 0,Y 601.406,Z 383.071,A -85,B 0,C 180,E1 -559.809,E2 -559.809} C_VEL
LIN {X 0,Y 601.404,Z 383.067,A -85,B 0,C 180,E1 -562.683,E2 -562.683} C_VEL
LIN {X 0,Y 601.402,Z 383.066,A -85,B 0,C 180,E1 -564.878,E2 -564.878} C_VEL
LIN {X 0,Y 601.419,Z 383.073,A -85,B 0,C 180,E1 -567.867,E2 -567.867} C_VEL
LIN {X 0,Y 601.441,Z 383.067,A -85,B 0,C 180,E1 -570.163,E2 -570.163} C_VEL
LIN {X 0,Y 601.415,Z 383.064,A -85,B 0,C 180,E1 -572.716,E2 -572.716} C_VEL
LIN {X 0,Y 601.41,Z 383.065,A -85,B 0,C 180,E1 -575.115,E2 -575.115} C_VEL
LIN {X 0,Y 601.429,Z 383.066,A -85,B 0,C 180,E1 -577.419,E2 -577.419} C_VEL
LIN {X 0,Y 601.407,Z 383.072,A -85,B 0,C 180,E1 -579.995,E2 -579.995} C_VEL
LIN {X 0,Y 601.405,Z 383.065,A -85,B 0,C 180,E1 -582.67,E2 -582.67} C_VEL
LIN {X 0,Y 601.418,Z 383.071,A -85,B 0,C 180,E1 -585.482,E2 -585.482} C_VEL
LIN {X 0,Y 601.422,Z 383.064,A -85,B 0,C 180,E1 -588.406,E2 -588.406} C_VEL
LIN {X 0,Y 601.429,Z 383.063,A -85,B 0,C 180,E1 -590.876,E2 -590.876} C_VEL
LIN {X 0,Y 601.437,Z 383.069,A -85,B 0,C 180,E1 -593.734,E2 -593.734} C_VEL
LIN {X 0,Y 601.427,Z 383.063,A -85,B 0,C 180,E1 -596.687,E2 -596.687} C_VEL
LIN {X 0,Y 601.424,Z 383.067,A -85,B 0,C 180,E1 -599.059,E2 -599.059} C_VEL
LIN {X 0,Y 601.432,Z 383.071,A -85,B 0,C 180,E1 -601.374,E2 -601.374} C_VEL
LIN {X 0,Y 601.414,Z 383.065,A -85,B 0,C 180,E1 -604.131,E2 -604.131} C_VEL
LIN {X 0,Y 601.417,Z 383.064,A -85,B 0,C 180,E1 -606.59,E2 -606.59} C_VEL
LIN {X 0,Y 601.429,Z 383.07,A -85,B 0,C 180,E1 -609.479,E2 -609.479} C_VEL
LIN {X 0,Y 601.393,Z 383.067,A -85,B 0,C 180,E1 -612.312,E2 -612.312} C_VEL
LIN {X 0,Y 601.41,Z 383.065,A -85,B 0,C 180,E1 -614.409,E2 -614.409} C_VEL
LIN {X 0,Y 601.417,Z 383.074,A -85,B 0,C 180,E1 -617.172,E2 -617.172} C_VEL
LIN {X 0,Y 601.439,Z 383.062,A -85,B 0,C 180,E1 -619.905,E2 -619.905} C_VEL
LIN {X 0,Y 601.437,Z 383.064,A -85,B 0,C 180,E1 -622.615,E2 -622.615} C_VEL
LIN {X 0,Y 601.417,Z 383.07,A -85,B 0,C 180,E1 -625.308,E2 -625.308} C_VEL
LIN {X 0,Y 601.437,Z 383.061,A -85,B 0,C 180,E1 -627.991,E2 -627.991} C_VEL
LIN {X 0,Y 601.446,Z 383.066,A -85,B 0,C 180,E1 -630.67,E2 -630.67} C_VEL
LIN {X 0,Y 601.426,Z 383.067,A -85,B 0,C 180,E1 -633.35,E2 -633.35} C_VEL
LIN {X 0,Y 601.441,Z 383.061,A -85,B 0,C 180,E1 -636.037,E2 -636.037} C_VEL
LIN {X 0,Y 601.432,Z 383.071,A -85,B 0,C 180,E1 -638.738,E2 -638.738} C_VEL
LIN {X 0,Y 601.431,Z 383.064,A -85,B 0,C 180,E1 -641.458,E2 -641.458} C_VEL
LIN {X 0,Y 601.416,Z 383.066,A -85,B 0,C 180,E1 -644.205,E2 -644.205} C_VEL
LIN {X 0,Y 601.429,Z 383.069,A -85,B 0,C 180,E1 -646.986,E2 -646.986} C_VEL
LIN {X 0,Y 601.402,Z 383.066,A -85,B 0,C 180,E1 -649.809,E2 -649.809} C_VEL
LIN {X 0,Y 601.412,Z 383.074,A -85,B 0,C 180,E1 -652.606,E2 -652.606} C_VEL
LIN {X 0,Y 601.401,Z 383.072,A -85,B 0,C 180,E1 -654.878,E2 -654.878} C_VEL
LIN {X 0,Y 601.418,Z 383.065,A -85,B 0,C 180,E1 -657.867,E2 -657.867} C_VEL
LIN {X 0,Y 601.423,Z 383.067,A -85,B 0,C 180,E1 -660.164,E2 -660.164} C_VEL
LIN {X 0,Y 601.425,Z 383.069,A -85,B 0,C 180,E1 -662.717,E2 -662.717} C_VEL
LIN {X 0,Y 601.406,Z 383.066,A -85,B 0,C 180,E1 -665.114,E2 -665.114} C_VEL
LIN {X 0,Y 601.43,Z 383.062,A -85,B 0,C 180,E1 -667.419,E2 -667.419} C_VEL
LIN {X 0,Y 601.406,Z 383.069,A -85,B 0,C 180,E1 -669.995,E2 -669.995} C_VEL
LIN {X 0,Y 601.434,Z 383.067,A -85,B 0,C 180,E1 -672.668,E2 -672.668} C_VEL
LIN {X 0,Y 601.42,Z 383.064,A -85,B 0,C 180,E1 -675.482,E2 -675.482} C_VEL
LIN {X 0,Y 601.421,Z 383.071,A -85,B 0,C 180,E1 -678.407,E2 -678.407} C_VEL
LIN {X 0,Y 601.435,Z 383.063,A -85,B 0,C 180,E1 -680.876,E2 -680.876} C_VEL
LIN {X 0,Y 601.44,Z 383.064,A -85,B 0,C 180,E1 -683.734,E2 -683.734} C_VEL
LIN {X 0,Y 601.429,Z 383.072,A -85,B 0,C 180,E1 -686.064,E2 -686.064} C_VEL
LIN {X 0,Y 601.428,Z 383.062,A -85,B 0,C 180,E1 -689.059,E2 -689.059} C_VEL
LIN {X 0,Y 601.426,Z 383.064,A -85,B 0,C 180,E1 -691.373,E2 -691.373} C_VEL
LIN {X 0,Y 601.401,Z 383.07,A -85,B 0,C 180,E1 -693.637,E2 -693.637} C_VEL
LIN {X 0,Y 601.417,Z 383.065,A -85,B 0,C 180,E1 -696.59,E2 -696.59} C_VEL
LIN {X 0,Y 601.425,Z 383.066,A -85,B 0,C 180,E1 -699.478,E2 -699.478} C_VEL
LIN {X 0,Y 601.399,Z 383.07,A -85,B 0,C 180,E1 -702.312,E2 -702.312} C_VEL
LIN {X 0,Y 601.416,Z 383.066,A -85,B 0,C 180,E1 -704.409,E2 -704.409} C_VEL
LIN {X 0,Y 601.421,Z 383.065,A -85,B 0,C 180,E1 -707.172,E2 -707.172} C_VEL
LIN {X 0,Y 601.43,Z 383.07,A -85,B 0,C 180,E1 -709.905,E2 -709.905} C_VEL
LIN {X 0,Y 601.449,Z 383.06,A -85,B 0,C 180,E1 -712.615,E2 -712.615} C_VEL
LIN {X 0,Y 601.422,Z 383.067,A -85,B 0,C 180,E1 -715.308,E2 -715.308} C_VEL
LIN {X 0,Y 601.423,Z 383.068,A -85,B 0,C 180,E1 -717.991,E2 -717.991} C_VEL
LIN {X 0,Y 601.448,Z 383.06,A -85,B 0,C 180,E1 -720.67,E2 -720.67} C_VEL
LIN {X 0,Y 601.428,Z 383.069,A -85,B 0,C 180,E1 -723.35,E2 -723.35} C_VEL
LIN {X 0,Y 601.41,Z 383.067,A -85,B 0,C 180,E1 -726.037,E2 -726.037} C_VEL
LIN {X 0,Y 601.435,Z 383.062,A -85,B 0,C 180,E1 -728.738,E2 -728.738} C_VEL
LIN {X 0,Y 601.432,Z 383.072,A -85,B 0,C 180,E1 -731.459,E2 -731.459} C_VEL
LIN {X 0,Y 601.416,Z 383.064,A -85,B 0,C 180,E1 -734.206,E2 -734.206} C_VEL
LIN {X 0,Y 601.431,Z 383.067,A -85,B 0,C 180,E1 -736.986,E2 -736.986} C_VEL
LIN {X 0,Y 601.409,Z 383.068,A -85,B 0,C 180,E1 -739.81,E2 -739.81} C_VEL
LIN {X 0,Y 601.409,Z 383.067,A -85,B 0,C 180,E1 -742.683,E2 -742.683} C_VEL
LIN {X 0,Y 601.404,Z 383.07,A -85,B 0,C 180,E1 -744.879,E2 -744.879} C_VEL
LIN {X 0,Y 601.42,Z 383.065,A -85,B 0,C 180,E1 -747.868,E2 -747.868} C_VEL
LIN {X 0,Y 601.427,Z 383.063,A -85,B 0,C 180,E1 -750.164,E2 -750.164} C_VEL
LIN {X 0,Y 601.417,Z 383.068,A -85,B 0,C 180,E1 -752.716,E2 -752.716} C_VEL
LIN {X 0,Y 601.413,Z 383.074,A -85,B 0,C 180,E1 -755.115,E2 -755.115} C_VEL
LIN {X 0,Y 601.435,Z 383.066,A -85,B 0,C 180,E1 -757.419,E2 -757.419} C_VEL
LIN {X 0,Y 601.411,Z 383.065,A -85,B 0,C 180,E1 -759.995,E2 -759.995} C_VEL
LIN {X 0,Y 601.411,Z 383.071,A -85,B 0,C 180,E1 -762.671,E2 -762.671} C_VEL
LIN {X 0,Y 601.426,Z 383.066,A -85,B 0,C 180,E1 -765.483,E2 -765.483} C_VEL
LIN {X 0,Y 601.433,Z 383.18,A -85,B 0,C 180,E1 -768.236,E2 -768.236} C_VEL
LIN {X 0,Y 601.468,Z 386.379,A -85,B 0,C 180,E1 -770.01,E2 -770.01} C_VEL
LIN {X 0,Y 601.447,Z 391.842,A -85,B 0,C 180,E1 -772.617,E2 -772.617} C_VEL
LIN {X 0,Y 601.445,Z 397.158,A -85,B 0,C 180,E1 -775.07,E2 -775.07} C_VEL
LIN {X 0,Y 601.46,Z 402.547,A -85,B 0,C 180,E1 -777.486,E2 -777.486} C_VEL
LIN {X 0,Y 601.431,Z 407.973,A -85,B 0,C 180,E1 -779.852,E2 -779.852} C_VEL
LIN {X 0,Y 601.4,Z 414.537,A -85,B 0,C 180,E1 -782.641,E2 -782.641} C_VEL
LIN {X 0,Y 601.399,Z 420.513,A -85,B 0,C 180,E1 -785.122,E2 -785.122} C_VEL
LIN {X 0,Y 601.387,Z 426.114,A -85,B 0,C 180,E1 -787.402,E2 -787.402} C_VEL
LIN {X 0,Y 601.374,Z 433.088,A -85,B 0,C 180,E1 -790.19,E2 -790.19} C_VEL
LIN {X 0,Y 601.356,Z 440.274,A -85,B 0,C 180,E1 -793.012,E2 -793.012} C_VEL
LIN {X 0,Y 601.35,Z 447.834,A -85,B 0,C 180,E1 -795.937,E2 -795.937} C_VEL
LIN {X 0,Y 601.368,Z 453.611,A -85,B 0,C 180,E1 -798.113,E2 -798.113} C_VEL
LIN {X 0,Y 601.598,Z 465.07,A -85,B 0,C 180,E1 -798.353,E2 -798.353} C_VEL
LIN {X 0,Y 601.549,Z 478.09,A -85,B 0,C 180,E1 -798.756,E2 -798.756} C_VEL
LIN {X 0,Y 601.513,Z 490.924,A -85,B 0,C 180,E1 -799.311,E2 -799.311} C_VEL
LIN {X 0,Y 601.477,Z 501.578,A -85,B 0,C 180,E1 -799.906,E2 -799.906} C_VEL
LIN {X 0,Y 601.449,Z 512.476,A -85,B 0,C 180,E1 -800.669,E2 -800.669} C_VEL
LIN {X 0,Y 601.429,Z 523.114,A -85,B 0,C 180,E1 -801.601,E2 -801.601} C_VEL
LIN {X 0,Y 601.418,Z 530.958,A -85,B 0,C 180,E1 -802.446,E2 -802.446} C_VEL
LIN {X 0,Y 601.37,Z 538.223,A -85,B 0,C 180,E1 -803.398,E2 -803.398} C_VEL
LIN {X 0,Y 601.372,Z 543.862,A -85,B 0,C 180,E1 -804.299,E2 -804.299} C_VEL
LIN {X 0,Y 601.336,Z 548.95,A -85,B 0,C 180,E1 -805.307,E2 -805.307} C_VEL
LIN {X 0,Y 601.367,Z 552.895,A -85,B 0,C 180,E1 -806.315,E2 -806.315} C_VEL
LIN {X 0,Y 601.325,Z 555.807,A -85,B 0,C 180,E1 -807.32,E2 -807.32} C_VEL
LIN {X 0,Y 601.343,Z 557.2,A -85,B 0,C 180,E1 -807.991,E2 -807.991} C_VEL
LIN {X 0,Y 601.339,Z 558.783,A -85,B 0,C 180,E1 -809.33,E2 -809.33} C_VEL
LIN {X 0,Y 601.335,Z 558.995,A -85,B 0,C 180,E1 -810,E2 -810} C_VEL
LIN {X 0,Y 601.348,Z 558.185,A -85,B 0,C 180,E1 -811.339,E2 -811.339} C_VEL
LIN {X 0,Y 601.343,Z 557.2,A -85,B 0,C 180,E1 -812.009,E2 -812.009} C_VEL
LIN {X 0,Y 601.325,Z 555.807,A -85,B 0,C 180,E1 -812.679,E2 -812.679} C_VEL
LIN {X 0,Y 601.367,Z 552.896,A -85,B 0,C 180,E1 -813.685,E2 -813.685} C_VEL
LIN {X 0,Y 601.336,Z 548.951,A -85,B 0,C 180,E1 -814.692,E2 -814.692} C_VEL
LIN {X 0,Y 601.372,Z 543.863,A -85,B 0,C 180,E1 -815.701,E2 -815.701} C_VEL
LIN {X 0,Y 601.382,Z 537.473,A -85,B 0,C 180,E1 -816.711,E2 -816.711} C_VEL
LIN {X 0,Y 601.396,Z 529.482,A -85,B 0,C 180,E1 -817.723,E2 -817.723} C_VEL
LIN {X 0,Y 601.423,Z 521.341,A -85,B 0,C 180,E1 -818.568,E2 -818.568} C_VEL
LIN {X 0,Y 601.455,Z 511.398,A -85,B 0,C 180,E1 -819.415,E2 -819.415} C_VEL
LIN {X 0,Y 601.491,Z 500.172,A -85,B 0,C 180,E1 -820.179,E2 -820.179} C_VEL
LIN {X 0,Y 601.534,Z 487.926,A -85,B 0,C 180,E1 -820.835,E2 -820.835} C_VEL
LIN {X 0,Y 601.563,Z 475.38,A -85,B 0,C 180,E1 -821.34,E2 -821.34} C_VEL
LIN {X 0,Y 601.607,Z 462.359,A -85,B 0,C 180,E1 -821.711,E2 -821.711} C_VEL
LIN {X 0,Y 601.368,Z 453.631,A -85,B 0,C 180,E1 -821.886,E2 -821.886} C_VEL
LIN {X 0,Y 601.361,Z 445.664,A -85,B 0,C 180,E1 -824.898,E2 -824.898} C_VEL
LIN {X 0,Y 601.359,Z 438.478,A -85,B 0,C 180,E1 -827.689,E2 -827.689} C_VEL
LIN {X 0,Y 601.374,Z 433.089,A -85,B 0,C 180,E1 -829.81,E2 -829.81} C_VEL
LIN {X 0,Y 601.396,Z 425.903,A -85,B 0,C 180,E1 -832.683,E2 -832.683} C_VEL
LIN {X 0,Y 601.418,Z 418.717,A -85,B 0,C 180,E1 -835.618,E2 -835.618} C_VEL
LIN {X 0,Y 601.434,Z 411.531,A -85,B 0,C 180,E1 -838.626,E2 -838.626} C_VEL
LIN {X 0,Y 601.442,Z 404.953,A -85,B 0,C 180,E1 -841.458,E2 -841.458} C_VEL
LIN {X 0,Y 601.429,Z 398.955,A -85,B 0,C 180,E1 -844.118,E2 -844.118} C_VEL
LIN {X 0,Y 601.443,Z 393.566,A -85,B 0,C 180,E1 -846.579,E2 -846.579} C_VEL
LIN {X 0,Y 601.468,Z 388.176,A -85,B 0,C 180,E1 -849.121,E2 -849.121} C_VEL
LIN {X 0,Y 601.517,Z 384.742,A -85,B 0,C 180,E1 -850.865,E2 -850.865} C_VEL
LIN {X 0,Y 601.446,Z 383.181,A -85,B 0,C 180,E1 -851.762,E2 -851.762} C_VEL
LIN {X 0,Y 601.422,Z 383.067,A -85,B 0,C 180,E1 -854.535,E2 -854.535} C_VEL
LIN {X 0,Y 601.409,Z 383.07,A -85,B 0,C 180,E1 -857.408,E2 -857.408} C_VEL
LIN {X 0,Y 601.409,Z 383.065,A -85,B 0,C 180,E1 -860.004,E2 -860.004} C_VEL
LIN {X 0,Y 601.435,Z 383.067,A -85,B 0,C 180,E1 -862.617,E2 -862.617} C_VEL
LIN {X 0,Y 601.437,Z 383.069,A -85,B 0,C 180,E1 -865.069,E2 -865.069} C_VEL
LIN {X 0,Y 601.422,Z 383.065,A -85,B 0,C 180,E1 -867.483,E2 -867.483} C_VEL
LIN {X 0,Y 601.445,Z 383.06,A -85,B 0,C 180,E1 -869.847,E2 -869.847} C_VEL
LIN {X 0,Y 601.455,Z 383.068,A -85,B 0,C 180,E1 -872.889,E2 -872.889} C_VEL
LIN {X 0,Y 601.459,Z 383.059,A -85,B 0,C 180,E1 -875.859,E2 -875.859} C_VEL
LIN {X 0,Y 601.406,Z 383.075,A -85,B 0,C 180,E1 -878.76,E2 -878.76} C_VEL
LIN {X 0,Y 601.416,Z 383.064,A -85,B 0,C 180,E1 -881.608,E2 -881.608} C_VEL
LIN {X 0,Y 601.415,Z 383.071,A -85,B 0,C 180,E1 -884.408,E2 -884.408} C_VEL
LIN {X 0,Y 601.421,Z 383.065,A -85,B 0,C 180,E1 -887.172,E2 -887.172} C_VEL
LIN {X 0,Y 601.43,Z 383.064,A -85,B 0,C 180,E1 -889.905,E2 -889.905} C_VEL
LIN {X 0,Y 601.448,Z 383.069,A -85,B 0,C 180,E1 -892.615,E2 -892.615} C_VEL
LIN {X 0,Y 601.423,Z 383.063,A -85,B 0,C 180,E1 -895.308,E2 -895.308} C_VEL
LIN {X 0,Y 601.423,Z 383.067,A -85,B 0,C 180,E1 -897.991,E2 -897.991} C_VEL
LIN {X 0,Y 601.447,Z 383.066,A -85,B 0,C 180,E1 -900.669,E2 -900.669} C_VEL
LIN {X 0,Y 601.427,Z 383.062,A -85,B 0,C 180,E1 -903.349,E2 -903.349} C_VEL
LIN {X 0,Y 601.409,Z 383.071,A -85,B 0,C 180,E1 -906.037,E2 -906.037} C_VEL
LIN {X 0,Y 601.435,Z 383.065,A -85,B 0,C 180,E1 -908.737,E2 -908.737} C_VEL
LIN {X 0,Y 601.43,Z 383.063,A -85,B 0,C 180,E1 -911.458,E2 -911.458} C_VEL
LIN {X 0,Y 601.406,Z 383.071,A -85,B 0,C 180,E1 -912.381,E2 -912.381} C_VEL
LIN {X 0,Y 600.744,Z 383.15,A -85,B 0,C 180,E1 -912.941,E2 -912.941} C_VEL
LIN {X 0,Y 597.893,Z 383.508,A -85,B 0,C 180,E1 -913.848,E2 -913.848} C_VEL
LIN {X 0,Y 595.481,Z 383.807,A -85,B 0,C 180,E1 -914.579,E2 -914.579} C_VEL
LIN {X 0,Y 594.444,Z 383.933,A -85,B 0,C 180,E1 -915.142,E2 -915.142} C_VEL
LIN {X 0,Y 594.359,Z 383.943,A -85,B 0,C 180,E1 -915.333,E2 -915.333} C_VEL
LIN {X 0,Y 594.378,Z 383.947,A -85,B 0,C 180,E1 -917.904,E2 -917.904} C_VEL
LIN {X 0,Y 594.372,Z 383.942,A -85,B 0,C 180,E1 -920.917,E2 -920.917} C_VEL
LIN {X 0,Y 594.388,Z 383.944,A -85,B 0,C 180,E1 -923.704,E2 -923.704} C_VEL
LIN {X 0,Y 594.384,Z 383.941,A -85,B 0,C 180,E1 -926.699,E2 -926.699} C_VEL
LIN {X 0,Y 594.375,Z 383.941,A -85,B 0,C 180,E1 -928.998,E2 -928.998} C_VEL
LIN {X 0,Y 594.386,Z 383.946,A -85,B 0,C 180,E1 -931.645,E2 -931.645} C_VEL
LIN {X 0,Y 594.392,Z 383.94,A -85,B 0,C 180,E1 -934.579,E2 -934.579} C_VEL
LIN {X 0,Y 594.38,Z 383.941,A -85,B 0,C 180,E1 -937.086,E2 -937.086} C_VEL
LIN {X 0,Y 594.373,Z 383.952,A -85,B 0,C 180,E1 -939.775,E2 -939.775} C_VEL
LIN {X 0,Y 594.362,Z 383.944,A -85,B 0,C 180,E1 -942.375,E2 -942.375} C_VEL
LIN {X 0,Y 594.355,Z 383.946,A -85,B 0,C 180,E1 -945.191,E2 -945.191} C_VEL
LIN {X 0,Y 594.383,Z 383.95,A -85,B 0,C 180,E1 -947.627,E2 -947.627} C_VEL
LIN {X 0,Y 594.385,Z 383.941,A -85,B 0,C 180,E1 -950.321,E2 -950.321} C_VEL
LIN {X 0,Y 594.38,Z 383.942,A -85,B 0,C 180,E1 -952.914,E2 -952.914} C_VEL
LIN {X 0,Y 594.38,Z 383.945,A -85,B 0,C 180,E1 -955.861,E2 -955.861} C_VEL
LIN {X 0,Y 594.385,Z 383.94,A -85,B 0,C 180,E1 -958.651,E2 -958.651} C_VEL
LIN {X 0,Y 594.38,Z 383.944,A -85,B 0,C 180,E1 -961.042,E2 -961.042} C_VEL
LIN {X 0,Y 594.387,Z 383.941,A -85,B 0,C 180,E1 -963.976,E2 -963.976} C_VEL
LIN {X 0,Y 594.386,Z 383.94,A -85,B 0,C 180,E1 -966.296,E2 -966.296} C_VEL
LIN {X 0,Y 594.403,Z 383.946,A -85,B 0,C 180,E1 -969.225,E2 -969.225} C_VEL
LIN {X 0,Y 594.351,Z 383.945,A -85,B 0,C 180,E1 -972.095,E2 -972.095} C_VEL
LIN {X 0,Y 594.363,Z 383.943,A -85,B 0,C 180,E1 -974.219,E2 -974.219} C_VEL
LIN {X 0,Y 594.364,Z 383.95,A -85,B 0,C 180,E1 -977.017,E2 -977.017} C_VEL
LIN {X 0,Y 594.397,Z 383.94,A -85,B 0,C 180,E1 -979.785,E2 -979.785} C_VEL
LIN {X 0,Y 594.391,Z 383.941,A -85,B 0,C 180,E1 -982.527,E2 -982.527} C_VEL
LIN {X 0,Y 594.388,Z 383.947,A -85,B 0,C 180,E1 -985.253,E2 -985.253} C_VEL
LIN {X 0,Y 594.405,Z 383.938,A -85,B 0,C 180,E1 -987.967,E2 -987.967} C_VEL
LIN {X 0,Y 594.417,Z 383.941,A -85,B 0,C 180,E1 -990.678,E2 -990.678} C_VEL
LIN {X 0,Y 594.378,Z 383.945,A -85,B 0,C 180,E1 -993.389,E2 -993.389} C_VEL
LIN {X 0,Y 594.394,Z 383.94,A -85,B 0,C 180,E1 -996.109,E2 -996.109} C_VEL
LIN {X 0,Y 594.394,Z 383.949,A -85,B 0,C 180,E1 -998.842,E2 -998.842} C_VEL
LIN {X 0,Y 594.391,Z 383.94,A -85,B 0,C 180,E1 -1001.596,E2 -1001.596} C_VEL
LIN {X 0,Y 594.386,Z 383.944,A -85,B 0,C 180,E1 -1004.377,E2 -1004.377} C_VEL
LIN {X 0,Y 594.387,Z 383.943,A -85,B 0,C 180,E1 -1007.193,E2 -1007.193} C_VEL
LIN {X 0,Y 594.372,Z 383.943,A -85,B 0,C 180,E1 -1010.054,E2 -1010.054} C_VEL
LIN {X 0,Y 594.361,Z 383.948,A -85,B 0,C 180,E1 -1012.967,E2 -1012.967} C_VEL
LIN {X 0,Y 594.376,Z 383.943,A -85,B 0,C 180,E1 -1015.193,E2 -1015.193} C_VEL
LIN {X 0,Y 594.381,Z 383.94,A -85,B 0,C 180,E1 -1017.527,E2 -1017.527} C_VEL
LIN {X 0,Y 594.383,Z 383.947,A -85,B 0,C 180,E1 -1020.328,E2 -1020.328} C_VEL
LIN {X 0,Y 594.377,Z 383.944,A -85,B 0,C 180,E1 -1022.95,E2 -1022.95} C_VEL
LIN {X 0,Y 594.377,Z 383.941,A -85,B 0,C 180,E1 -1025.407,E2 -1025.407} C_VEL
LIN {X 0,Y 594.382,Z 383.943,A -85,B 0,C 180,E1 -1027.941,E2 -1027.941} C_VEL
LIN {X 0,Y 594.377,Z 383.944,A -85,B 0,C 180,E1 -1030.823,E2 -1030.823} C_VEL
LIN {X 0,Y 594.382,Z 383.94,A -85,B 0,C 180,E1 -1033.298,E2 -1033.298} C_VEL
LIN {X 0,Y 594.363,Z 383.951,A -85,B 0,C 180,E1 -1036.16,E2 -1036.16} C_VEL
LIN {X 0,Y 594.378,Z 383.946,A -85,B 0,C 180,E1 -1038.537,E2 -1038.537} C_VEL
LIN {X 0,Y 594.384,Z 383.94,A -85,B 0,C 180,E1 -1041.295,E2 -1041.295} C_VEL
LIN {X 0,Y 594.392,Z 383.943,A -85,B 0,C 180,E1 -1043.759,E2 -1043.759} C_VEL
LIN {X 0,Y 594.376,Z 383.95,A -85,B 0,C 180,E1 -1046.239,E2 -1046.239} C_VEL
LIN {X 0,Y 594.386,Z 383.942,A -85,B 0,C 180,E1 -1048.651,E2 -1048.651} C_VEL
LIN {X 0,Y 594.378,Z 383.941,A -85,B 0,C 180,E1 -1051.042,E2 -1051.042} C_VEL
LIN {X 0,Y 594.385,Z 383.941,A -85,B 0,C 180,E1 -1053.301,E2 -1053.301} C_VEL
LIN {X 0,Y 594.389,Z 383.944,A -85,B 0,C 180,E1 -1056.296,E2 -1056.296} C_VEL
LIN {X 0,Y 594.397,Z 383.939,A -85,B 0,C 180,E1 -1059.225,E2 -1059.225} C_VEL
LIN {X 0,Y 594.378,Z 383.947,A -85,B 0,C 180,E1 -1062.096,E2 -1062.096} C_VEL
LIN {X 0,Y 594.369,Z 383.946,A -85,B 0,C 180,E1 -1064.22,E2 -1064.22} C_VEL
LIN {X 0,Y 594.369,Z 383.942,A -85,B 0,C 180,E1 -1067.017,E2 -1067.017} C_VEL
LIN {X 0,Y 594.39,Z 383.95,A -85,B 0,C 180,E1 -1069.784,E2 -1069.784} C_VEL
LIN {X 0,Y 594.398,Z 383.939,A -85,B 0,C 180,E1 -1072.527,E2 -1072.527} C_VEL
LIN {X 0,Y 594.391,Z 383.942,A -85,B 0,C 180,E1 -1075.253,E2 -1075.253} C_VEL
LIN {X 0,Y 594.393,Z 383.944,A -85,B 0,C 180,E1 -1077.968,E2 -1077.968} C_VEL
LIN {X 0,Y 594.419,Z 383.936,A -85,B 0,C 180,E1 -1080.678,E2 -1080.678} C_VEL
LIN {X 0,Y 594.38,Z 383.948,A -85,B 0,C 180,E1 -1083.39,E2 -1083.39} C_VEL
LIN {X 0,Y 594.366,Z 383.944,A -85,B 0,C 180,E1 -1086.109,E2 -1086.109} C_VEL
LIN {X 0,Y 594.397,Z 383.94,A -85,B 0,C 180,E1 -1088.842,E2 -1088.842} C_VEL
LIN {X 0,Y 594.391,Z 383.947,A -85,B 0,C 180,E1 -1091.596,E2 -1091.596} C_VEL
LIN {X 0,Y 594.386,Z 383.94,A -85,B 0,C 180,E1 -1094.377,E2 -1094.377} C_VEL
LIN {X 0,Y 594.389,Z 383.947,A -85,B 0,C 180,E1 -1097.194,E2 -1097.194} C_VEL
LIN {X 0,Y 594.375,Z 383.942,A -85,B 0,C 180,E1 -1100.054,E2 -1100.054} C_VEL
LIN {X 0,Y 594.362,Z 383.948,A -85,B 0,C 180,E1 -1102.968,E2 -1102.968} C_VEL
LIN {X 0,Y 594.376,Z 383.951,A -85,B 0,C 180,E1 -1105.193,E2 -1105.193} C_VEL
LIN {X 0,Y 594.383,Z 383.945,A -85,B 0,C 180,E1 -1107.527,E2 -1107.527} C_VEL
LIN {X 0,Y 594.386,Z 383.94,A -85,B 0,C 180,E1 -1110.329,E2 -1110.329} C_VEL
LIN {X 0,Y 594.376,Z 383.949,A -85,B 0,C 180,E1 -1112.951,E2 -1112.951} C_VEL
LIN {X 0,Y 594.382,Z 383.945,A -85,B 0,C 180,E1 -1115.407,E2 -1115.407} C_VEL
LIN {X 0,Y 594.386,Z 383.94,A -85,B 0,C 180,E1 -1117.941,E2 -1117.941} C_VEL
LIN {X 0,Y 594.379,Z 383.949,A -85,B 0,C 180,E1 -1120.823,E2 -1120.823} C_VEL
LIN {X 0,Y 594.367,Z 383.943,A -85,B 0,C 180,E1 -1123.84,E2 -1123.84} C_VEL
LIN {X 0,Y 594.381,Z 383.95,A -85,B 0,C 180,E1 -1126.702,E2 -1126.702} C_VEL
LIN {X 0,Y 594.374,Z 383.947,A -85,B 0,C 180,E1 -1127.626,E2 -1127.626} C_VEL
LIN {X 0,Y 594.513,Z 385.036,A -85,B 0,C 180,E1 -1128.548,E2 -1128.548} C_VEL
LIN {X 0,Y 594.474,Z 390.143,A -85,B 0,C 180,E1 -1131.285,E2 -1131.285} C_VEL
LIN {X 0,Y 594.421,Z 395.361,A -85,B 0,C 180,E1 -1133.761,E2 -1133.761} C_VEL
LIN {X 0,Y 594.397,Z 400.751,A -85,B 0,C 180,E1 -1136.24,E2 -1136.24} C_VEL
LIN {X 0,Y 594.396,Z 406.141,A -85,B 0,C 180,E1 -1138.652,E2 -1138.652} C_VEL
LIN {X 0,Y 594.383,Z 411.625,A -85,B 0,C 180,E1 -1141.043,E2 -1141.043} C_VEL
LIN {X 0,Y 594.344,Z 418.716,A -85,B 0,C 180,E1 -1144.055,E2 -1144.055} C_VEL
LIN {X 0,Y 594.313,Z 424.106,A -85,B 0,C 180,E1 -1146.293,E2 -1146.293} C_VEL
LIN {X 0,Y 594.332,Z 431.292,A -85,B 0,C 180,E1 -1149.222,E2 -1149.222} C_VEL
LIN {X 0,Y 594.304,Z 436.681,A -85,B 0,C 180,E1 -1151.38,E2 -1151.38} C_VEL
LIN {X 0,Y 594.262,Z 443.867,A -85,B 0,C 180,E1 -1154.216,E2 -1154.216} C_VEL
LIN {X 0,Y 594.26,Z 449.257,A -85,B 0,C 180,E1 -1156.318,E2 -1156.318} C_VEL
LIN {X 0,Y 594.28,Z 453.593,A -85,B 0,C 180,E1 -1157.969,E2 -1157.969} C_VEL
LIN {X 0,Y 594.658,Z 458.384,A -85,B 0,C 180,E1 -1158.064,E2 -1158.064} C_VEL
LIN {X 0,Y 594.644,Z 470.506,A -85,B 0,C 180,E1 -1158.366,E2 -1158.366} C_VEL
LIN {X 0,Y 594.56,Z 482.301,A -85,B 0,C 180,E1 -1158.788,E2 -1158.788} C_VEL
LIN {X 0,Y 594.514,Z 494.204,A -85,B 0,C 180,E1 -1159.356,E2 -1159.356} C_VEL
LIN {X 0,Y 594.475,Z 505.476,A -85,B 0,C 180,E1 -1160.044,E2 -1160.044} C_VEL
LIN {X 0,Y 594.406,Z 515.645,A -85,B 0,C 180,E1 -1160.815,E2 -1160.815} C_VEL
LIN {X 0,Y 594.372,Z 524.778,A -85,B 0,C 180,E1 -1161.672,E2 -1161.672} C_VEL
LIN {X 0,Y 594.317,Z 533.683,A -85,B 0,C 180,E1 -1162.697,E2 -1162.697} C_VEL
LIN {X 0,Y 594.281,Z 540.167,A -85,B 0,C 180,E1 -1163.615,E2 -1163.615} C_VEL
LIN {X 0,Y 594.289,Z 545.68,A -85,B 0,C 180,E1 -1164.571,E2 -1164.571} C_VEL
LIN {X 0,Y 594.27,Z 550.373,A -85,B 0,C 180,E1 -1165.591,E2 -1165.591} C_VEL
LIN {X 0,Y 594.267,Z 553.958,A -85,B 0,C 180,E1 -1166.61,E2 -1166.61} C_VEL
LIN {X 0,Y 594.226,Z 555.805,A -85,B 0,C 180,E1 -1167.288,E2 -1167.288} C_VEL
LIN {X 0,Y 594.242,Z 557.199,A -85,B 0,C 180,E1 -1167.967,E2 -1167.967} C_VEL
LIN {X 0,Y 594.239,Z 558.783,A -85,B 0,C 180,E1 -1169.322,E2 -1169.322} C_VEL
LIN {X 0,Y 594.236,Z 558.991,A -85,B 0,C 180,E1 -1170,E2 -1170} C_VEL
LIN {X 0,Y 594.248,Z 558.186,A -85,B 0,C 180,E1 -1171.355,E2 -1171.355} C_VEL
LIN {X 0,Y 594.242,Z 557.199,A -85,B 0,C 180,E1 -1172.033,E2 -1172.033} C_VEL
LIN {X 0,Y 594.225,Z 555.805,A -85,B 0,C 180,E1 -1172.711,E2 -1172.711} C_VEL
LIN {X 0,Y 594.288,Z 552.895,A -85,B 0,C 180,E1 -1173.729,E2 -1173.729} C_VEL
LIN {X 0,Y 594.241,Z 548.95,A -85,B 0,C 180,E1 -1174.749,E2 -1174.749} C_VEL
LIN {X 0,Y 594.298,Z 543.859,A -85,B 0,C 180,E1 -1175.769,E2 -1175.769} C_VEL
LIN {X 0,Y 594.316,Z 537.472,A -85,B 0,C 180,E1 -1176.791,E2 -1176.791} C_VEL
LIN {X 0,Y 594.346,Z 529.484,A -85,B 0,C 180,E1 -1177.815,E2 -1177.815} C_VEL
LIN {X 0,Y 594.377,Z 521.343,A -85,B 0,C 180,E1 -1178.671,E2 -1178.671} C_VEL
LIN {X 0,Y 594.419,Z 511.391,A -85,B 0,C 180,E1 -1179.528,E2 -1179.528} C_VEL
LIN {X 0,Y 594.464,Z 500.172,A -85,B 0,C 180,E1 -1180.3,E2 -1180.3} C_VEL
LIN {X 0,Y 594.557,Z 487.748,A -85,B 0,C 180,E1 -1180.972,E2 -1180.972} C_VEL
LIN {X 0,Y 594.589,Z 475.698,A -85,B 0,C 180,E1 -1181.464,E2 -1181.464} C_VEL
LIN {X 0,Y 594.663,Z 463.268,A -85,B 0,C 180,E1 -1181.828,E2 -1181.828} C_VEL
LIN {X 0,Y 594.406,Z 454.61,A -85,B 0,C 180,E1 -1182.011,E2 -1182.011} C_VEL
LIN {X 0,Y 594.285,Z 453.468,A -85,B 0,C 180,E1 -1182.052,E2 -1182.052} C_VEL
LIN {X 0,Y 594.277,Z 445.664,A -85,B 0,C 180,E1 -1185.08,E2 -1185.08} C_VEL
LIN {X 0,Y 594.289,Z 440.275,A -85,B 0,C 180,E1 -1187.196,E2 -1187.196} C_VEL
LIN {X 0,Y 594.289,Z 434.885,A -85,B 0,C 180,E1 -1189.337,E2 -1189.337} C_VEL
LIN {X 0,Y 594.292,Z 429.496,A -85,B 0,C 180,E1 -1191.506,E2 -1191.506} C_VEL
LIN {X 0,Y 594.312,Z 424.106,A -85,B 0,C 180,E1 -1193.707,E2 -1193.707} C_VEL
LIN {X 0,Y 594.341,Z 418.555,A -85,B 0,C 180,E1 -1196.013,E2 -1196.013} C_VEL
LIN {X 0,Y 594.38,Z 411.531,A -85,B 0,C 180,E1 -1198.998,E2 -1198.998} C_VEL
LIN {X 0,Y 594.397,Z 405.47,A -85,B 0,C 180,E1 -1201.645,E2 -1201.645} C_VEL
LIN {X 0,Y 594.399,Z 399.913,A -85,B 0,C 180,E1 -1204.14,E2 -1204.14} C_VEL
LIN {X 0,Y 594.43,Z 394.827,A -85,B 0,C 180,E1 -1206.489,E2 -1206.489} C_VEL
LIN {X 0,Y 594.471,Z 389.973,A -85,B 0,C 180,E1 -1208.797,E2 -1208.797} C_VEL
LIN {X 0,Y 594.512,Z 385.038,A -85,B 0,C 180,E1 -1211.452,E2 -1211.452} C_VEL
LIN {X 0,Y 594.376,Z 383.949,A -85,B 0,C 180,E1 -1212.374,E2 -1212.374} C_VEL
LIN {X 0,Y 594.362,Z 383.952,A -85,B 0,C 180,E1 -1215.19,E2 -1215.19} C_VEL
LIN {X 0,Y 594.381,Z 383.941,A -85,B 0,C 180,E1 -1218.151,E2 -1218.151} C_VEL
LIN {X 0,Y 594.386,Z 383.947,A -85,B 0,C 180,E1 -1221.195,E2 -1221.195} C_VEL
LIN {X 0,Y 594.394,Z 383.94,A -85,B 0,C 180,E1 -1223.758,E2 -1223.758} C_VEL
LIN {X 0,Y 594.377,Z 383.942,A -85,B 0,C 180,E1 -1226.238,E2 -1226.238} C_VEL
LIN {X 0,Y 594.388,Z 383.946,A -85,B 0,C 180,E1 -1228.65,E2 -1228.65} C_VEL
LIN {X 0,Y 594.379,Z 383.947,A -85,B 0,C 180,E1 -1231.041,E2 -1231.041} C_VEL
LIN {X 0,Y 594.385,Z 383.943,A -85,B 0,C 180,E1 -1233.3,E2 -1233.3} C_VEL
LIN {X 0,Y 594.389,Z 383.942,A -85,B 0,C 180,E1 -1236.296,E2 -1236.296} C_VEL
LIN {X 0,Y 594.397,Z 383.941,A -85,B 0,C 180,E1 -1239.224,E2 -1239.224} C_VEL
LIN {X 0,Y 594.378,Z 383.943,A -85,B 0,C 180,E1 -1242.095,E2 -1242.095} C_VEL
LIN {X 0,Y 594.368,Z 383.946,A -85,B 0,C 180,E1 -1244.219,E2 -1244.219} C_VEL
LIN {X 0,Y 594.369,Z 383.945,A -85,B 0,C 180,E1 -1247.017,E2 -1247.017} C_VEL
LIN {X 0,Y 594.39,Z 383.94,A -85,B 0,C 180,E1 -1249.784,E2 -1249.784} C_VEL
LIN {X 0,Y 594.397,Z 383.949,A -85,B 0,C 180,E1 -1252.527,E2 -1252.527} C_VEL
LIN {X 0,Y 594.392,Z 383.939,A -85,B 0,C 180,E1 -1255.252,E2 -1255.252} C_VEL
LIN {X 0,Y 594.393,Z 383.942,A -85,B 0,C 180,E1 -1257.967,E2 -1257.967} C_VEL
LIN {X 0,Y 594.418,Z 383.941,A -85,B 0,C 180,E1 -1260.677,E2 -1260.677} C_VEL
LIN {X 0,Y 594.379,Z 383.941,A -85,B 0,C 180,E1 -1263.389,E2 -1263.389} C_VEL
LIN {X 0,Y 594.365,Z 383.949,A -85,B 0,C 180,E1 -1266.109,E2 -1266.109} C_VEL
LIN {X 0,Y 594.396,Z 383.94,A -85,B 0,C 180,E1 -1268.842,E2 -1268.842} C_VEL
LIN {X 0,Y 594.388,Z 383.941,A -85,B 0,C 180,E1 -1271.595,E2 -1271.595} C_VEL
LIN {X 0,Y 594.382,Z 383.947,A -85,B 0,C 180,E1 -1274.377,E2 -1274.377} C_VEL
LIN {X 0,Y 594.359,Z 383.943,A -85,B 0,C 180,E1 -1275.333,E2 -1275.333} C_VEL
LIN {X 0,Y 593.691,Z 384.034,A -85,B 0,C 180,E1 -1275.899,E2 -1275.899} C_VEL
LIN {X 0,Y 590.838,Z 384.394,A -85,B 0,C 180,E1 -1276.817,E2 -1276.817} C_VEL
LIN {X 0,Y 588.432,Z 384.695,A -85,B 0,C 180,E1 -1277.556,E2 -1277.556} C_VEL
LIN {X 0,Y 587.402,Z 384.82,A -85,B 0,C 180,E1 -1278.126,E2 -1278.126} C_VEL
LIN {X 0,Y 587.32,Z 384.827,A -85,B 0,C 180,E1 -1278.319,E2 -1278.319} C_VEL
LIN {X 0,Y 587.321,Z 384.82,A -85,B 0,C 180,E1 -1281.037,E2 -1281.037} C_VEL
LIN {X 0,Y 587.317,Z 384.821,A -85,B 0,C 180,E1 -1283.258,E2 -1283.258} C_VEL
LIN {X 0,Y 587.33,Z 384.822,A -85,B 0,C 180,E1 -1285.516,E2 -1285.516} C_VEL
LIN {X 0,Y 587.341,Z 384.825,A -85,B 0,C 180,E1 -1287.818,E2 -1287.818} C_VEL
LIN {X 0,Y 587.344,Z 384.819,A -85,B 0,C 180,E1 -1290.513,E2 -1290.513} C_VEL
LIN {X 0,Y 587.329,Z 384.822,A -85,B 0,C 180,E1 -1293.396,E2 -1293.396} C_VEL
LIN {X 0,Y 587.351,Z 384.826,A -85,B 0,C 180,E1 -1295.895,E2 -1295.895} C_VEL
LIN {X 0,Y 587.328,Z 384.82,A -85,B 0,C 180,E1 -1298.479,E2 -1298.479} C_VEL
LIN {X 0,Y 587.331,Z 384.82,A -85,B 0,C 180,E1 -1301.157,E2 -1301.157} C_VEL
LIN {X 0,Y 587.327,Z 384.823,A -85,B 0,C 180,E1 -1304.114,E2 -1304.114} C_VEL
LIN {X 0,Y 587.331,Z 384.82,A -85,B 0,C 180,E1 -1306.996,E2 -1306.996} C_VEL
LIN {X 0,Y 587.316,Z 384.825,A -85,B 0,C 180,E1 -1309.981,E2 -1309.981} C_VEL
LIN {X 0,Y 587.339,Z 384.818,A -85,B 0,C 180,E1 -1312.393,E2 -1312.393} C_VEL
LIN {X 0,Y 587.343,Z 384.819,A -85,B 0,C 180,E1 -1314.946,E2 -1314.946} C_VEL
LIN {X 0,Y 587.338,Z 384.827,A -85,B 0,C 180,E1 -1317.422,E2 -1317.422} C_VEL
LIN {X 0,Y 587.329,Z 384.823,A -85,B 0,C 180,E1 -1319.83,E2 -1319.83} C_VEL
LIN {X 0,Y 587.347,Z 384.817,A -85,B 0,C 180,E1 -1322.307,E2 -1322.307} C_VEL
LIN {X 0,Y 587.335,Z 384.818,A -85,B 0,C 180,E1 -1324.484,E2 -1324.484} C_VEL
LIN {X 0,Y 587.336,Z 384.826,A -85,B 0,C 180,E1 -1327.487,E2 -1327.487} C_VEL
LIN {X 0,Y 587.339,Z 384.818,A -85,B 0,C 180,E1 -1330.425,E2 -1330.425} C_VEL
LIN {X 0,Y 587.347,Z 384.827,A -85,B 0,C 180,E1 -1333.311,E2 -1333.311} C_VEL
LIN {X 0,Y 587.356,Z 384.816,A -85,B 0,C 180,E1 -1336.155,E2 -1336.155} C_VEL
LIN {X 0,Y 587.34,Z 384.824,A -85,B 0,C 180,E1 -1338.963,E2 -1338.963} C_VEL
LIN {X 0,Y 587.367,Z 384.816,A -85,B 0,C 180,E1 -1341.745,E2 -1341.745} C_VEL
LIN {X 0,Y 587.362,Z 384.817,A -85,B 0,C 180,E1 -1344.507,E2 -1344.507} C_VEL
LIN {X 0,Y 587.369,Z 384.821,A -85,B 0,C 180,E1 -1347.257,E2 -1347.257} C_VEL
LIN {X 0,Y 587.382,Z 384.813,A -85,B 0,C 180,E1 -1350,E2 -1350} C_VEL
LIN {X 0,Y 587.369,Z 384.821,A -85,B 0,C 180,E1 -1352.743,E2 -1352.743} C_VEL
LIN {X 0,Y 587.362,Z 384.817,A -85,B 0,C 180,E1 -1355.493,E2 -1355.493} C_VEL
LIN {X 0,Y 587.367,Z 384.816,A -85,B 0,C 180,E1 -1358.255,E2 -1358.255} C_VEL
LIN {X 0,Y 587.345,Z 384.822,A -85,B 0,C 180,E1 -1361.134,E2 -1361.134} C_VEL
LIN {X 0,Y 587.362,Z 384.818,A -85,B 0,C 180,E1 -1364.261,E2 -1364.261} C_VEL
LIN {X 0,Y 587.347,Z 384.818,A -85,B 0,C 180,E1 -1367.406,E2 -1367.406} C_VEL
LIN {X 0,Y 587.328,Z 384.823,A -85,B 0,C 180,E1 -1370.305,E2 -1370.305} C_VEL
LIN {X 0,Y 587.319,Z 384.822,A -85,B 0,C 180,E1 -1373.259,E2 -1373.259} C_VEL
LIN {X 0,Y 587.335,Z 384.818,A -85,B 0,C 180,E1 -1375.516,E2 -1375.516} C_VEL
LIN {X 0,Y 587.346,Z 384.817,A -85,B 0,C 180,E1 -1377.818,E2 -1377.818} C_VEL
LIN {X 0,Y 587.337,Z 384.828,A -85,B 0,C 180,E1 -1380.511,E2 -1380.511} C_VEL
LIN {X 0,Y 587.337,Z 384.819,A -85,B 0,C 180,E1 -1383.112,E2 -1383.112} C_VEL
LIN {X 0,Y 587.351,Z 384.818,A -85,B 0,C 180,E1 -1385.895,E2 -1385.895} C_VEL
LIN {X 0,Y 587.328,Z 384.828,A -85,B 0,C 180,E1 -1388.479,E2 -1388.479} C_VEL
LIN {X 0,Y 587.333,Z 384.819,A -85,B 0,C 180,E1 -1391.157,E2 -1391.157} C_VEL
LIN {X 0,Y 587.329,Z 384.826,A -85,B 0,C 180,E1 -1394.114,E2 -1394.114} C_VEL
LIN {X 0,Y 587.309,Z 384.822,A -85,B 0,C 180,E1 -1396.994,E2 -1396.994} C_VEL
LIN {X 0,Y 587.315,Z 384.823,A -85,B 0,C 180,E1 -1399.746,E2 -1399.746} C_VEL
LIN {X 0,Y 587.34,Z 384.824,A -85,B 0,C 180,E1 -1402.393,E2 -1402.393} C_VEL
LIN {X 0,Y 587.346,Z 384.817,A -85,B 0,C 180,E1 -1404.946,E2 -1404.946} C_VEL
LIN {X 0,Y 587.333,Z 384.819,A -85,B 0,C 180,E1 -1407.421,E2 -1407.421} C_VEL
LIN {X 0,Y 587.342,Z 384.823,A -85,B 0,C 180,E1 -1409.831,E2 -1409.831} C_VEL
LIN {X 0,Y 587.346,Z 384.822,A -85,B 0,C 180,E1 -1412.307,E2 -1412.307} C_VEL
LIN {X 0,Y 587.332,Z 384.821,A -85,B 0,C 180,E1 -1414.484,E2 -1414.484} C_VEL
LIN {X 0,Y 587.313,Z 384.821,A -85,B 0,C 180,E1 -1417.131,E2 -1417.131} C_VEL
LIN {X 0,Y 587.327,Z 384.825,A -85,B 0,C 180,E1 -1419.696,E2 -1419.696} C_VEL
LIN {X 0,Y 587.355,Z 384.816,A -85,B 0,C 180,E1 -1422.595,E2 -1422.595} C_VEL
LIN {X 0,Y 587.36,Z 384.824,A -85,B 0,C 180,E1 -1425.739,E2 -1425.739} C_VEL
LIN {X 0,Y 587.339,Z 384.821,A -85,B 0,C 180,E1 -1428.263,E2 -1428.263} C_VEL
LIN {X 0,Y 587.341,Z 384.818,A -85,B 0,C 180,E1 -1431.051,E2 -1431.051} C_VEL
LIN {X 0,Y 587.371,Z 384.817,A -85,B 0,C 180,E1 -1433.264,E2 -1433.264} C_VEL
LIN {X 0,Y 587.313,Z 384.827,A -85,B 0,C 180,E1 -1435.883,E2 -1435.883} C_VEL
LIN {X 0,Y 587.363,Z 384.82,A -85,B 0,C 180,E1 -1437.943,E2 -1437.943} C_VEL
LIN {X 0,Y 587.389,Z 384.811,A -85,B 0,C 180,E1 -1440.686,E2 -1440.686} C_VEL
LIN {X 0,Y 587.331,Z 384.827,A -85,B 0,C 180,E1 -1443.43,E2 -1443.43} C_VEL
LIN {X 0,Y 587.357,Z 384.825,A -85,B 0,C 180,E1 -1445.493,E2 -1445.493} C_VEL
LIN {X 0,Y 587.367,Z 384.815,A -85,B 0,C 180,E1 -1448.256,E2 -1448.256} C_VEL
LIN {X 0,Y 587.344,Z 384.822,A -85,B 0,C 180,E1 -1451.134,E2 -1451.134} C_VEL
LIN {X 0,Y 587.362,Z 384.815,A -85,B 0,C 180,E1 -1454.261,E2 -1454.261} C_VEL
LIN {X 0,Y 587.355,Z 384.825,A -85,B 0,C 180,E1 -1457.406,E2 -1457.406} C_VEL
LIN {X 0,Y 587.328,Z 384.819,A -85,B 0,C 180,E1 -1460.305,E2 -1460.305} C_VEL
LIN {X 0,Y 587.321,Z 384.83,A -85,B 0,C 180,E1 -1463.259,E2 -1463.259} C_VEL
LIN {X 0,Y 587.333,Z 384.823,A -85,B 0,C 180,E1 -1465.517,E2 -1465.517} C_VEL
LIN {X 0,Y 587.346,Z 384.818,A -85,B 0,C 180,E1 -1467.818,E2 -1467.818} C_VEL
LIN {X 0,Y 587.341,Z 384.819,A -85,B 0,C 180,E1 -1470.512,E2 -1470.512} C_VEL
LIN {X 0,Y 587.333,Z 384.823,A -85,B 0,C 180,E1 -1473.397,E2 -1473.397} C_VEL
LIN {X 0,Y 587.356,Z 384.816,A -85,B 0,C 180,E1 -1475.896,E2 -1475.896} C_VEL
LIN {X 0,Y 587.333,Z 384.821,A -85,B 0,C 180,E1 -1478.48,E2 -1478.48} C_VEL
LIN {X 0,Y 587.337,Z 384.826,A -85,B 0,C 180,E1 -1481.157,E2 -1481.157} C_VEL
LIN {X 0,Y 587.326,Z 384.821,A -85,B 0,C 180,E1 -1484.114,E2 -1484.114} C_VEL
LIN {X 0,Y 587.324,Z 384.829,A -85,B 0,C 180,E1 -1486.995,E2 -1486.995} C_VEL
LIN {X 0,Y 587.419,Z 385.379,A -85,B 0,C 180,E1 -1487.934,E2 -1487.934} C_VEL
LIN {X 0,Y 587.51,Z 388.881,A -85,B 0,C 180,E1 -1489.96,E2 -1489.96} C_VEL
LIN {X 0,Y 587.411,Z 393.565,A -85,B 0,C 180,E1 -1492.398,E2 -1492.398} C_VEL
LIN {X 0,Y 587.386,Z 398.954,A -85,B 0,C 180,E1 -1494.949,E2 -1494.949} C_VEL
LIN {X 0,Y 587.374,Z 404.344,A -85,B 0,C 180,E1 -1497.424,E2 -1497.424} C_VEL
LIN {X 0,Y 587.335,Z 409.734,A -85,B 0,C 180,E1 -1499.83,E2 -1499.83} C_VEL
LIN {X 0,Y 587.299,Z 415.442,A -85,B 0,C 180,E1 -1502.318,E2 -1502.318} C_VEL
LIN {X 0,Y 587.295,Z 422.309,A -85,B 0,C 180,E1 -1505.239,E2 -1505.239} C_VEL
LIN {X 0,Y 587.248,Z 429.495,A -85,B 0,C 180,E1 -1508.223,E2 -1508.223} C_VEL
LIN {X 0,Y 587.256,Z 436.681,A -85,B 0,C 180,E1 -1511.148,E2 -1511.148} C_VEL
LIN {X 0,Y 587.194,Z 443.867,A -85,B 0,C 180,E1 -1514.021,E2 -1514.021} C_VEL
LIN {X 0,Y 587.193,Z 449.257,A -85,B 0,C 180,E1 -1516.15,E2 -1516.15} C_VEL
LIN {X 0,Y 587.167,Z 453.567,A -85,B 0,C 180,E1 -1517.821,E2 -1517.821} C_VEL
LIN {X 0,Y 587.733,Z 458.388,A -85,B 0,C 180,E1 -1517.921,E2 -1517.921} C_VEL
LIN {X 0,Y 587.687,Z 470.508,A -85,B 0,C 180,E1 -1518.226,E2 -1518.226} C_VEL
LIN {X 0,Y 587.588,Z 483.255,A -85,B 0,C 180,E1 -1518.695,E2 -1518.695} C_VEL
LIN {X 0,Y 587.537,Z 495.77,A -85,B 0,C 180,E1 -1519.315,E2 -1519.315} C_VEL
LIN {X 0,Y 587.463,Z 506.748,A -85,B 0,C 180,E1 -1520.01,E2 -1520.01} C_VEL
LIN {X 0,Y 587.357,Z 517.589,A -85,B 0,C 180,E1 -1520.878,E2 -1520.878} C_VEL
LIN {X 0,Y 587.301,Z 526.4,A -85,B 0,C 180,E1 -1521.744,E2 -1521.744} C_VEL
LIN {X 0,Y 587.232,Z 535.002,A -85,B 0,C 180,E1 -1522.781,E2 -1522.781} C_VEL
LIN {X 0,Y 587.212,Z 541.868,A -85,B 0,C 180,E1 -1523.816,E2 -1523.816} C_VEL
LIN {X 0,Y 587.167,Z 547.364,A -85,B 0,C 180,E1 -1524.85,E2 -1524.85} C_VEL
LIN {X 0,Y 587.182,Z 551.67,A -85,B 0,C 180,E1 -1525.882,E2 -1525.882} C_VEL
LIN {X 0,Y 587.193,Z 553.96,A -85,B 0,C 180,E1 -1526.569,E2 -1526.569} C_VEL
LIN {X 0,Y 587.132,Z 555.802,A -85,B 0,C 180,E1 -1527.256,E2 -1527.256} C_VEL
LIN {X 0,Y 587.141,Z 557.196,A -85,B 0,C 180,E1 -1527.942,E2 -1527.942} C_VEL
LIN {X 0,Y 587.147,Z 558.186,A -85,B 0,C 180,E1 -1528.628,E2 -1528.628} C_VEL
LIN {X 0,Y 587.137,Z 558.987,A -85,B 0,C 180,E1 -1530,E2 -1530} C_VEL
LIN {X 0,Y 587.147,Z 558.187,A -85,B 0,C 180,E1 -1531.372,E2 -1531.372} C_VEL
LIN {X 0,Y 587.141,Z 557.197,A -85,B 0,C 180,E1 -1532.058,E2 -1532.058} C_VEL
LIN {X 0,Y 587.132,Z 555.803,A -85,B 0,C 180,E1 -1532.744,E2 -1532.744} C_VEL
LIN {X 0,Y 587.212,Z 552.893,A -85,B 0,C 180,E1 -1533.774,E2 -1533.774} C_VEL
LIN {X 0,Y 587.147,Z 548.947,A -85,B 0,C 180,E1 -1534.806,E2 -1534.806} C_VEL
LIN {X 0,Y 587.229,Z 543.854,A -85,B 0,C 180,E1 -1535.838,E2 -1535.838} C_VEL
LIN {X 0,Y 587.23,Z 537.469,A -85,B 0,C 180,E1 -1536.873,E2 -1536.873} C_VEL
LIN {X 0,Y 587.287,Z 529.485,A -85,B 0,C 180,E1 -1537.91,E2 -1537.91} C_VEL
LIN {X 0,Y 587.336,Z 521.345,A -85,B 0,C 180,E1 -1538.775,E2 -1538.775} C_VEL
LIN {X 0,Y 587.392,Z 511.385,A -85,B 0,C 180,E1 -1539.643,E2 -1539.643} C_VEL
LIN {X 0,Y 587.462,Z 501.572,A -85,B 0,C 180,E1 -1540.337,E2 -1540.337} C_VEL
LIN {X 0,Y 587.549,Z 490.935,A -85,B 0,C 180,E1 -1540.946,E2 -1540.946} C_VEL
LIN {X 0,Y 587.63,Z 478.419,A -85,B 0,C 180,E1 -1541.501,E2 -1541.501} C_VEL
LIN {X 0,Y 587.692,Z 465.923,A -85,B 0,C 180,E1 -1541.904,E2 -1541.904} C_VEL
LIN {X 0,Y 587.574,Z 456.121,A -85,B 0,C 180,E1 -1542.126,E2 -1542.126} C_VEL
LIN {X 0,Y 587.163,Z 453.468,A -85,B 0,C 180,E1 -1542.2,E2 -1542.2} C_VEL
LIN {X 0,Y 587.206,Z 447.461,A -85,B 0,C 180,E1 -1544.556,E2 -1544.556} C_VEL
LIN {X 0,Y 587.212,Z 440.275,A -85,B 0,C 180,E1 -1547.41,E2 -1547.41} C_VEL
LIN {X 0,Y 587.215,Z 434.885,A -85,B 0,C 180,E1 -1549.579,E2 -1549.579} C_VEL
LIN {X 0,Y 587.248,Z 429.496,A -85,B 0,C 180,E1 -1551.777,E2 -1551.777} C_VEL
LIN {X 0,Y 587.294,Z 422.31,A -85,B 0,C 180,E1 -1554.761,E2 -1554.761} C_VEL
LIN {X 0,Y 587.298,Z 415.442,A -85,B 0,C 180,E1 -1557.682,E2 -1557.682} C_VEL
LIN {X 0,Y 587.334,Z 409.734,A -85,B 0,C 180,E1 -1560.169,E2 -1560.169} C_VEL
LIN {X 0,Y 587.394,Z 403.146,A -85,B 0,C 180,E1 -1563.119,E2 -1563.119} C_VEL
LIN {X 0,Y 587.413,Z 397.159,A -85,B 0,C 180,E1 -1565.891,E2 -1565.891} C_VEL
LIN {X 0,Y 587.479,Z 390.866,A -85,B 0,C 180,E1 -1568.959,E2 -1568.959} C_VEL
LIN {X 0,Y 587.541,Z 386.9,A -85,B 0,C 180,E1 -1571.139,E2 -1571.139} C_VEL
LIN {X 0,Y 587.395,Z 385.304,A -85,B 0,C 180,E1 -1572.114,E2 -1572.114} C_VEL
LIN {X 0,Y 587.325,Z 384.829,A -85,B 0,C 180,E1 -1573.119,E2 -1573.119} C_VEL
LIN {X 0,Y 587.32,Z 384.821,A -85,B 0,C 180,E1 -1576.049,E2 -1576.049} C_VEL
LIN {X 0,Y 587.335,Z 384.828,A -85,B 0,C 180,E1 -1578.924,E2 -1578.924} C_VEL
LIN {X 0,Y 587.331,Z 384.822,A -85,B 0,C 180,E1 -1581.52,E2 -1581.52} C_VEL
LIN {X 0,Y 587.349,Z 384.82,A -85,B 0,C 180,E1 -1584.454,E2 -1584.454} C_VEL
LIN {X 0,Y 587.335,Z 384.829,A -85,B 0,C 180,E1 -1586.887,E2 -1586.887} C_VEL
LIN {X 0,Y 587.348,Z 384.818,A -85,B 0,C 180,E1 -1589.487,E2 -1589.487} C_VEL
LIN {X 0,Y 587.347,Z 384.819,A -85,B 0,C 180,E1 -1592.306,E2 -1592.306} C_VEL
LIN {X 0,Y 587.333,Z 384.824,A -85,B 0,C 180,E1 -1594.483,E2 -1594.483} C_VEL
LIN {X 0,Y 587.314,Z 384.825,A -85,B 0,C 180,E1 -1597.13,E2 -1597.13} C_VEL
LIN {X 0,Y 587.327,Z 384.819,A -85,B 0,C 180,E1 -1599.695,E2 -1599.695} C_VEL
LIN {X 0,Y 587.355,Z 384.825,A -85,B 0,C 180,E1 -1602.594,E2 -1602.594} C_VEL
LIN {X 0,Y 587.359,Z 384.815,A -85,B 0,C 180,E1 -1605.739,E2 -1605.739} C_VEL
LIN {X 0,Y 587.338,Z 384.823,A -85,B 0,C 180,E1 -1608.263,E2 -1608.263} C_VEL
LIN {X 0,Y 587.341,Z 384.82,A -85,B 0,C 180,E1 -1611.051,E2 -1611.051} C_VEL
LIN {X 0,Y 587.369,Z 384.814,A -85,B 0,C 180,E1 -1613.263,E2 -1613.263} C_VEL
LIN {X 0,Y 587.313,Z 384.823,A -85,B 0,C 180,E1 -1615.882,E2 -1615.882} C_VEL
LIN {X 0,Y 587.363,Z 384.817,A -85,B 0,C 180,E1 -1617.942,E2 -1617.942} C_VEL
LIN {X 0,Y 587.388,Z 384.817,A -85,B 0,C 180,E1 -1620.685,E2 -1620.685} C_VEL
LIN {X 0,Y 587.33,Z 384.819,A -85,B 0,C 180,E1 -1623.43,E2 -1623.43} C_VEL
LIN {X 0,Y 587.356,Z 384.816,A -85,B 0,C 180,E1 -1625.493,E2 -1625.493} C_VEL
LIN {X 0,Y 587.365,Z 384.825,A -85,B 0,C 180,E1 -1628.255,E2 -1628.255} C_VEL
LIN {X 0,Y 587.339,Z 384.818,A -85,B 0,C 180,E1 -1631.133,E2 -1631.133} C_VEL
LIN {X 0,Y 587.356,Z 384.82,A -85,B 0,C 180,E1 -1633.845,E2 -1633.845} C_VEL
LIN {X 0,Y 587.355,Z 384.816,A -85,B 0,C 180,E1 -1636.819,E2 -1636.819} C_VEL
LIN {X 0,Y 587.32,Z 384.827,A -85,B 0,C 180,E1 -1638.319,E2 -1638.319} C_VEL
LIN {X 0,Y 586.664,Z 384.904,A -85,B 0,C 180,E1 -1638.891,E2 -1638.891} C_VEL
LIN {X 0,Y 583.829,Z 385.261,A -85,B 0,C 180,E1 -1639.819,E2 -1639.819} C_VEL
LIN {X 0,Y 581.419,Z 385.558,A -85,B 0,C 180,E1 -1640.566,E2 -1640.566} C_VEL
LIN {X 0,Y 580.368,Z 385.686,A -85,B 0,C 180,E1 -1641.142,E2 -1641.142} C_VEL
LIN {X 0,Y 580.275,Z 385.698,A -85,B 0,C 180,E1 -1641.338,E2 -1641.338} C_VEL
LIN {X 0,Y 580.295,Z 385.7,A -85,B 0,C 180,E1 -1644.316,E2 -1644.316} C_VEL
LIN {X 0,Y 580.303,Z 385.695,A -85,B 0,C 180,E1 -1646.622,E2 -1646.622} C_VEL
LIN {X 0,Y 580.299,Z 385.696,A -85,B 0,C 180,E1 -1649.311,E2 -1649.311} C_VEL
LIN {X 0,Y 580.295,Z 385.7,A -85,B 0,C 180,E1 -1652.2,E2 -1652.2} C_VEL
LIN {X 0,Y 580.295,Z 385.695,A -85,B 0,C 180,E1 -1654.695,E2 -1654.695} C_VEL
LIN {X 0,Y 580.294,Z 385.697,A -85,B 0,C 180,E1 -1657.268,E2 -1657.268} C_VEL
LIN {X 0,Y 580.293,Z 385.698,A -85,B 0,C 180,E1 -1660.272,E2 -1660.272} C_VEL
LIN {X 0,Y 580.274,Z 385.698,A -85,B 0,C 180,E1 -1662.706,E2 -1662.706} C_VEL
LIN {X 0,Y 580.267,Z 385.708,A -85,B 0,C 180,E1 -1665.609,E2 -1665.609} C_VEL
LIN {X 0,Y 580.308,Z 385.695,A -85,B 0,C 180,E1 -1668.235,E2 -1668.235} C_VEL
LIN {X 0,Y 580.283,Z 385.698,A -85,B 0,C 180,E1 -1670.966,E2 -1670.966} C_VEL
LIN {X 0,Y 580.29,Z 385.706,A -85,B 0,C 180,E1 -1673.599,E2 -1673.599} C_VEL
LIN {X 0,Y 580.315,Z 385.694,A -85,B 0,C 180,E1 -1676.146,E2 -1676.146} C_VEL
LIN {X 0,Y 580.284,Z 385.697,A -85,B 0,C 180,E1 -1678.616,E2 -1678.616} C_VEL
LIN {X 0,Y 580.29,Z 385.699,A -85,B 0,C 180,E1 -1681.024,E2 -1681.024} C_VEL
LIN {X 0,Y 580.323,Z 385.697,A -85,B 0,C 180,E1 -1683.659,E2 -1683.659} C_VEL
LIN {X 0,Y 580.275,Z 385.698,A -85,B 0,C 180,E1 -1686.442,E2 -1686.442} C_VEL
LIN {X 0,Y 580.272,Z 385.706,A -85,B 0,C 180,E1 -1689.438,E2 -1689.438} C_VEL
LIN {X 0,Y 580.265,Z 385.704,A -85,B 0,C 180,E1 -1691.645,E2 -1691.645} C_VEL
LIN {X 0,Y 580.275,Z 385.7,A -85,B 0,C 180,E1 -1693.826,E2 -1693.826} C_VEL
LIN {X 0,Y 580.322,Z 385.693,A -85,B 0,C 180,E1 -1695.983,E2 -1695.983} C_VEL
LIN {X 0,Y 580.301,Z 385.699,A -85,B 0,C 180,E1 -1698.827,E2 -1698.827} C_VEL
LIN {X 0,Y 580.331,Z 385.694,A -85,B 0,C 180,E1 -1701.644,E2 -1701.644} C_VEL
LIN {X 0,Y 580.33,Z 385.693,A -85,B 0,C 180,E1 -1704.441,E2 -1704.441} C_VEL
LIN {X 0,Y 580.344,Z 385.69,A -85,B 0,C 180,E1 -1707.918,E2 -1707.918} C_VEL
LIN {X 0,Y 580.359,Z 385.693,A -85,B 0,C 180,E1 -1710.694,E2 -1710.694} C_VEL
LIN {X 0,Y 580.281,Z 385.7,A -85,B 0,C 180,E1 -1713.472,E2 -1713.472} C_VEL
LIN {X 0,Y 580.33,Z 385.693,A -85,B 0,C 180,E1 -1715.56,E2 -1715.56} C_VEL
LIN {X 0,Y 580.331,Z 385.694,A -85,B 0,C 180,E1 -1718.356,E2 -1718.356} C_VEL
LIN {X 0,Y 580.297,Z 385.7,A -85,B 0,C 180,E1 -1721.191,E2 -1721.191} C_VEL
LIN {X 0,Y 580.323,Z 385.693,A -85,B 0,C 180,E1 -1724.017,E2 -1724.017} C_VEL
LIN {X 0,Y 580.309,Z 385.701,A -85,B 0,C 180,E1 -1726.914,E2 -1726.914} C_VEL
LIN {X 0,Y 580.302,Z 385.694,A -85,B 0,C 180,E1 -1729.822,E2 -1729.822} C_VEL
LIN {X 0,Y 580.292,Z 385.703,A -85,B 0,C 180,E1 -1732.802,E2 -1732.802} C_VEL
LIN {X 0,Y 580.305,Z 385.697,A -85,B 0,C 180,E1 -1735.08,E2 -1735.08} C_VEL
LIN {X 0,Y 580.316,Z 385.693,A -85,B 0,C 180,E1 -1737.863,E2 -1737.863} C_VEL
LIN {X 0,Y 580.288,Z 385.703,A -85,B 0,C 180,E1 -1740.696,E2 -1740.696} C_VEL
LIN {X 0,Y 580.302,Z 385.694,A -85,B 0,C 180,E1 -1743.317,E2 -1743.317} C_VEL
LIN {X 0,Y 580.32,Z 385.693,A -85,B 0,C 180,E1 -1745.767,E2 -1745.767} C_VEL
LIN {X 0,Y 580.284,Z 385.702,A -85,B 0,C 180,E1 -1748.146,E2 -1748.146} C_VEL
LIN {X 0,Y 580.296,Z 385.698,A -85,B 0,C 180,E1 -1750.843,E2 -1750.843} C_VEL
LIN {X 0,Y 580.286,Z 385.697,A -85,B 0,C 180,E1 -1753.657,E2 -1753.657} C_VEL
LIN {X 0,Y 580.271,Z 385.703,A -85,B 0,C 180,E1 -1756.609,E2 -1756.609} C_VEL
LIN {X 0,Y 580.296,Z 385.695,A -85,B 0,C 180,E1 -1759.157,E2 -1759.157} C_VEL
LIN {X 0,Y 580.286,Z 385.702,A -85,B 0,C 180,E1 -1761.927,E2 -1761.927} C_VEL
LIN {X 0,Y 580.302,Z 385.699,A -85,B 0,C 180,E1 -1764.457,E2 -1764.457} C_VEL
LIN {X 0,Y 580.286,Z 385.696,A -85,B 0,C 180,E1 -1766.975,E2 -1766.975} C_VEL
LIN {X 0,Y 580.305,Z 385.695,A -85,B 0,C 180,E1 -1769.426,E2 -1769.426} C_VEL
LIN {X 0,Y 580.314,Z 385.701,A -85,B 0,C 180,E1 -1772.137,E2 -1772.137} C_VEL
LIN {X 0,Y 580.317,Z 385.693,A -85,B 0,C 180,E1 -1775.27,E2 -1775.27} C_VEL
LIN {X 0,Y 580.27,Z 385.709,A -85,B 0,C 180,E1 -1777.948,E2 -1777.948} C_VEL
LIN {X 0,Y 580.313,Z 385.693,A -85,B 0,C 180,E1 -1780.914,E2 -1780.914} C_VEL
LIN {X 0,Y 580.279,Z 385.707,A -85,B 0,C 180,E1 -1783.826,E2 -1783.826} C_VEL
LIN {X 0,Y 580.323,Z 385.699,A -85,B 0,C 180,E1 -1785.983,E2 -1785.983} C_VEL
LIN {X 0,Y 580.299,Z 385.695,A -85,B 0,C 180,E1 -1788.827,E2 -1788.827} C_VEL
LIN {X 0,Y 580.33,Z 385.699,A -85,B 0,C 180,E1 -1791.644,E2 -1791.644} C_VEL
LIN {X 0,Y 580.322,Z 385.692,A -85,B 0,C 180,E1 -1794.441,E2 -1794.441} C_VEL
LIN {X 0,Y 580.34,Z 385.693,A -85,B 0,C 180,E1 -1797.224,E2 -1797.224} C_VEL
LIN {X 0,Y 580.348,Z 385.692,A -85,B 0,C 180,E1 -1800,E2 -1800} C_VEL
LIN {X 0,Y 580.34,Z 385.69,A -85,B 0,C 180,E1 -1802.777,E2 -1802.777} C_VEL
LIN {X 0,Y 580.323,Z 385.702,A -85,B 0,C 180,E1 -1805.56,E2 -1805.56} C_VEL
LIN {X 0,Y 580.331,Z 385.691,A -85,B 0,C 180,E1 -1808.356,E2 -1808.356} C_VEL
LIN {X 0,Y 580.296,Z 385.701,A -85,B 0,C 180,E1 -1811.192,E2 -1811.192} C_VEL
LIN {X 0,Y 580.324,Z 385.693,A -85,B 0,C 180,E1 -1814.017,E2 -1814.017} C_VEL
LIN {X 0,Y 580.309,Z 385.697,A -85,B 0,C 180,E1 -1816.914,E2 -1816.914} C_VEL
LIN {X 0,Y 580.304,Z 385.696,A -85,B 0,C 180,E1 -1819.823,E2 -1819.823} C_VEL
LIN {X 0,Y 580.292,Z 385.698,A -85,B 0,C 180,E1 -1822.803,E2 -1822.803} C_VEL
LIN {X 0,Y 580.305,Z 385.702,A -85,B 0,C 180,E1 -1825.08,E2 -1825.08} C_VEL
LIN {X 0,Y 580.299,Z 385.695,A -85,B 0,C 180,E1 -1828.186,E2 -1828.186} C_VEL
LIN {X 0,Y 580.292,Z 385.699,A -85,B 0,C 180,E1 -1830.697,E2 -1830.697} C_VEL
LIN {X 0,Y 580.302,Z 385.701,A -85,B 0,C 180,E1 -1833.317,E2 -1833.317} C_VEL
LIN {X 0,Y 580.325,Z 385.693,A -85,B 0,C 180,E1 -1835.768,E2 -1835.768} C_VEL
LIN {X 0,Y 580.288,Z 385.697,A -85,B 0,C 180,E1 -1838.147,E2 -1838.147} C_VEL
LIN {X 0,Y 580.3,Z 385.704,A -85,B 0,C 180,E1 -1840.844,E2 -1840.844} C_VEL
LIN {X 0,Y 580.278,Z 385.7,A -85,B 0,C 180,E1 -1843.658,E2 -1843.658} C_VEL
LIN {X 0,Y 580.287,Z 385.705,A -85,B 0,C 180,E1 -1846.609,E2 -1846.609} C_VEL
LIN {X 0,Y 580.27,Z 385.707,A -85,B 0,C 180,E1 -1847.294,E2 -1847.294} C_VEL
LIN {X 0,Y 580.567,Z 388.788,A -85,B 0,C 180,E1 -1849.18,E2 -1849.18} C_VEL
LIN {X 0,Y 580.442,Z 393.756,A -85,B 0,C 180,E1 -1851.908,E2 -1851.908} C_VEL
LIN {X 0,Y 580.393,Z 398.954,A -85,B 0,C 180,E1 -1854.463,E2 -1854.463} C_VEL
LIN {X 0,Y 580.351,Z 404.344,A -85,B 0,C 180,E1 -1856.979,E2 -1856.979} C_VEL
LIN {X 0,Y 580.305,Z 409.734,A -85,B 0,C 180,E1 -1859.426,E2 -1859.426} C_VEL
LIN {X 0,Y 580.247,Z 415.899,A -85,B 0,C 180,E1 -1862.152,E2 -1862.152} C_VEL
LIN {X 0,Y 580.232,Z 422.309,A -85,B 0,C 180,E1 -1864.917,E2 -1864.917} C_VEL
LIN {X 0,Y 580.199,Z 429.495,A -85,B 0,C 180,E1 -1867.945,E2 -1867.945} C_VEL
LIN {X 0,Y 580.183,Z 436.681,A -85,B 0,C 180,E1 -1870.91,E2 -1870.91} C_VEL
LIN {X 0,Y 580.13,Z 443.867,A -85,B 0,C 180,E1 -1873.821,E2 -1873.821} C_VEL
LIN {X 0,Y 580.091,Z 451.053,A -85,B 0,C 180,E1 -1876.692,E2 -1876.692} C_VEL
LIN {X 0,Y 580.091,Z 453.54,A -85,B 0,C 180,E1 -1877.671,E2 -1877.671} C_VEL
LIN {X 0,Y 580.801,Z 458.392,A -85,B 0,C 180,E1 -1877.775,E2 -1877.775} C_VEL
LIN {X 0,Y 580.744,Z 470.509,A -85,B 0,C 180,E1 -1878.084,E2 -1878.084} C_VEL
LIN {X 0,Y 580.628,Z 482.281,A -85,B 0,C 180,E1 -1878.515,E2 -1878.515} C_VEL
LIN {X 0,Y 580.548,Z 494.203,A -85,B 0,C 180,E1 -1879.097,E2 -1879.097} C_VEL
LIN {X 0,Y 580.452,Z 505.479,A -85,B 0,C 180,E1 -1879.8,E2 -1879.8} C_VEL
LIN {X 0,Y 580.352,Z 515.643,A -85,B 0,C 180,E1 -1880.591,E2 -1880.591} C_VEL
LIN {X 0,Y 580.279,Z 524.771,A -85,B 0,C 180,E1 -1881.468,E2 -1881.468} C_VEL
LIN {X 0,Y 580.199,Z 533.677,A -85,B 0,C 180,E1 -1882.518,E2 -1882.518} C_VEL
LIN {X 0,Y 580.11,Z 541.286,A -85,B 0,C 180,E1 -1883.639,E2 -1883.639} C_VEL
LIN {X 0,Y 580.086,Z 547.364,A -85,B 0,C 180,E1 -1884.787,E2 -1884.787} C_VEL
LIN {X 0,Y 580.105,Z 551.669,A -85,B 0,C 180,E1 -1885.831,E2 -1885.831} C_VEL
LIN {X 0,Y 580.123,Z 553.961,A -85,B 0,C 180,E1 -1886.527,E2 -1886.527} C_VEL
LIN {X 0,Y 580.043,Z 555.8,A -85,B 0,C 180,E1 -1887.222,E2 -1887.222} C_VEL
LIN {X 0,Y 580.047,Z 558.187,A -85,B 0,C 180,E1 -1888.611,E2 -1888.611} C_VEL
LIN {X 0,Y 580.04,Z 558.782,A -85,B 0,C 180,E1 -1889.306,E2 -1889.306} C_VEL
LIN {X 0,Y 580.037,Z 558.983,A -85,B 0,C 180,E1 -1890,E2 -1890} C_VEL
LIN {X 0,Y 580.04,Z 558.783,A -85,B 0,C 180,E1 -1890.694,E2 -1890.694} C_VEL
LIN {X 0,Y 580.047,Z 558.187,A -85,B 0,C 180,E1 -1891.388,E2 -1891.388} C_VEL
LIN {X 0,Y 580.043,Z 555.8,A -85,B 0,C 180,E1 -1892.778,E2 -1892.778} C_VEL
LIN {X 0,Y 580.109,Z 552.89,A -85,B 0,C 180,E1 -1893.82,E2 -1893.82} C_VEL
LIN {X 0,Y 580.053,Z 548.944,A -85,B 0,C 180,E1 -1894.865,E2 -1894.865} C_VEL
LIN {X 0,Y 580.161,Z 543.849,A -85,B 0,C 180,E1 -1895.91,E2 -1895.91} C_VEL
LIN {X 0,Y 580.157,Z 537.466,A -85,B 0,C 180,E1 -1896.958,E2 -1896.958} C_VEL
LIN {X 0,Y 580.242,Z 529.487,A -85,B 0,C 180,E1 -1898.007,E2 -1898.007} C_VEL
LIN {X 0,Y 580.305,Z 521.346,A -85,B 0,C 180,E1 -1898.883,E2 -1898.883} C_VEL
LIN {X 0,Y 580.373,Z 511.379,A -85,B 0,C 180,E1 -1899.76,E2 -1899.76} C_VEL
LIN {X 0,Y 580.477,Z 501.564,A -85,B 0,C 180,E1 -1900.463,E2 -1900.463} C_VEL
LIN {X 0,Y 580.56,Z 490.937,A -85,B 0,C 180,E1 -1901.079,E2 -1901.079} C_VEL
LIN {X 0,Y 580.656,Z 478.145,A -85,B 0,C 180,E1 -1901.652,E2 -1901.652} C_VEL
LIN {X 0,Y 580.748,Z 465.034,A -85,B 0,C 180,E1 -1902.071,E2 -1902.071} C_VEL
LIN {X 0,Y 580.562,Z 456.509,A -85,B 0,C 180,E1 -1902.267,E2 -1902.267} C_VEL
LIN {X 0,Y 580.094,Z 453.468,A -85,B 0,C 180,E1 -1902.351,E2 -1902.351} C_VEL
LIN {X 0,Y 580.123,Z 447.461,A -85,B 0,C 180,E1 -1904.738,E2 -1904.738} C_VEL
LIN {X 0,Y 580.143,Z 440.275,A -85,B 0,C 180,E1 -1907.629,E2 -1907.629} C_VEL
LIN {X 0,Y 580.16,Z 434.885,A -85,B 0,C 180,E1 -1909.827,E2 -1909.827} C_VEL
LIN {X 0,Y 580.199,Z 429.496,A -85,B 0,C 180,E1 -1912.055,E2 -1912.055} C_VEL
LIN {X 0,Y 580.231,Z 422.31,A -85,B 0,C 180,E1 -1915.083,E2 -1915.083} C_VEL
LIN {X 0,Y 580.245,Z 415.9,A -85,B 0,C 180,E1 -1917.848,E2 -1917.848} C_VEL
LIN {X 0,Y 580.304,Z 409.734,A -85,B 0,C 180,E1 -1920.574,E2 -1920.574} C_VEL
LIN {X 0,Y 580.358,Z 403.686,A -85,B 0,C 180,E1 -1923.324,E2 -1923.324} C_VEL
LIN {X 0,Y 580.386,Z 397.159,A -85,B 0,C 180,E1 -1926.394,E2 -1926.394} C_VEL
LIN {X 0,Y 580.494,Z 391.691,A -85,B 0,C 180,E1 -1929.209,E2 -1929.209} C_VEL
LIN {X 0,Y 580.551,Z 387.87,A -85,B 0,C 180,E1 -1931.361,E2 -1931.361} C_VEL
LIN {X 0,Y 580.269,Z 385.708,A -85,B 0,C 180,E1 -1932.706,E2 -1932.706} C_VEL
LIN {X 0,Y 580.268,Z 385.703,A -85,B 0,C 180,E1 -1935.608,E2 -1935.608} C_VEL
LIN {X 0,Y 580.312,Z 385.695,A -85,B 0,C 180,E1 -1938.234,E2 -1938.234} C_VEL
LIN {X 0,Y 580.289,Z 385.706,A -85,B 0,C 180,E1 -1940.966,E2 -1940.966} C_VEL
LIN {X 0,Y 580.294,Z 385.697,A -85,B 0,C 180,E1 -1943.598,E2 -1943.598} C_VEL
LIN {X 0,Y 580.316,Z 385.693,A -85,B 0,C 180,E1 -1946.145,E2 -1946.145} C_VEL
LIN {X 0,Y 580.286,Z 385.702,A -85,B 0,C 180,E1 -1948.615,E2 -1948.615} C_VEL
LIN {X 0,Y 580.29,Z 385.703,A -85,B 0,C 180,E1 -1951.023,E2 -1951.023} C_VEL
LIN {X 0,Y 580.288,Z 385.696,A -85,B 0,C 180,E1 -1953.665,E2 -1953.665} C_VEL
LIN {X 0,Y 580.297,Z 385.695,A -85,B 0,C 180,E1 -1955.683,E2 -1955.683} C_VEL
LIN {X 0,Y 580.27,Z 385.699,A -85,B 0,C 180,E1 -1957.947,E2 -1957.947} C_VEL
LIN {X 0,Y 580.313,Z 385.699,A -85,B 0,C 180,E1 -1960.914,E2 -1960.914} C_VEL
LIN {X 0,Y 580.278,Z 385.698,A -85,B 0,C 180,E1 -1963.825,E2 -1963.825} C_VEL
LIN {X 0,Y 580.322,Z 385.693,A -85,B 0,C 180,E1 -1965.983,E2 -1965.983} C_VEL
LIN {X 0,Y 580.298,Z 385.7,A -85,B 0,C 180,E1 -1968.826,E2 -1968.826} C_VEL
LIN {X 0,Y 580.329,Z 385.691,A -85,B 0,C 180,E1 -1971.644,E2 -1971.644} C_VEL
LIN {X 0,Y 580.322,Z 385.702,A -85,B 0,C 180,E1 -1974.44,E2 -1974.44} C_VEL
LIN {X 0,Y 580.339,Z 385.69,A -85,B 0,C 180,E1 -1977.223,E2 -1977.223} C_VEL
LIN {X 0,Y 580.346,Z 385.693,A -85,B 0,C 180,E1 -1980,E2 -1980} C_VEL
LIN {X 0,Y 580.339,Z 385.693,A -85,B 0,C 180,E1 -1982.776,E2 -1982.776} C_VEL
LIN {X 0,Y 580.322,Z 385.692,A -85,B 0,C 180,E1 -1985.559,E2 -1985.559} C_VEL
LIN {X 0,Y 580.328,Z 385.7,A -85,B 0,C 180,E1 -1988.356,E2 -1988.356} C_VEL
LIN {X 0,Y 580.291,Z 385.695,A -85,B 0,C 180,E1 -1991.191,E2 -1991.191} C_VEL
LIN {X 0,Y 580.32,Z 385.699,A -85,B 0,C 180,E1 -1994.017,E2 -1994.017} C_VEL
LIN {X 0,Y 580.306,Z 385.694,A -85,B 0,C 180,E1 -1996.915,E2 -1996.915} C_VEL
LIN {X 0,Y 580.3,Z 385.7,A -85,B 0,C 180,E1 -1999.822,E2 -1999.822} C_VEL
LIN {X 0,Y 580.275,Z 385.698,A -85,B 0,C 180,E1 -2001.338,E2 -2001.338} C_VEL
LIN {X 0,Y 579.581,Z 385.792,A -85,B 0,C 180,E1 -2001.917,E2 -2001.917} C_VEL
LIN {X 0,Y 576.705,Z 386.148,A -85,B 0,C 180,E1 -2002.857,E2 -2002.857} C_VEL
LIN {X 0,Y 574.31,Z 386.446,A -85,B 0,C 180,E1 -2003.613,E2 -2003.613} C_VEL
LIN {X 0,Y 573.311,Z 386.572,A -85,B 0,C 180,E1 -2004.197,E2 -2004.197} C_VEL
LIN {X 0,Y 573.244,Z 386.575,A -85,B 0,C 180,E1 -2004.394,E2 -2004.394} C_VEL
LIN {X 0,Y 573.26,Z 386.571,A -85,B 0,C 180,E1 -2006.975,E2 -2006.975} C_VEL
LIN {X 0,Y 573.246,Z 386.576,A -85,B 0,C 180,E1 -2009.49,E2 -2009.49} C_VEL
LIN {X 0,Y 573.248,Z 386.578,A -85,B 0,C 180,E1 -2012.229,E2 -2012.229} C_VEL
LIN {X 0,Y 573.245,Z 386.573,A -85,B 0,C 180,E1 -2014.774,E2 -2014.774} C_VEL
LIN {X 0,Y 573.247,Z 386.574,A -85,B 0,C 180,E1 -2017.166,E2 -2017.166} C_VEL
LIN {X 0,Y 573.243,Z 386.581,A -85,B 0,C 180,E1 -2019.607,E2 -2019.607} C_VEL
LIN {X 0,Y 573.236,Z 386.574,A -85,B 0,C 180,E1 -2022.642,E2 -2022.642} C_VEL
LIN {X 0,Y 573.232,Z 386.585,A -85,B 0,C 180,E1 -2025.667,E2 -2025.667} C_VEL
LIN {X 0,Y 573.239,Z 386.574,A -85,B 0,C 180,E1 -2028.545,E2 -2028.545} C_VEL
LIN {X 0,Y 573.242,Z 386.579,A -85,B 0,C 180,E1 -2031.299,E2 -2031.299} C_VEL
LIN {X 0,Y 573.258,Z 386.575,A -85,B 0,C 180,E1 -2034.011,E2 -2034.011} C_VEL
LIN {X 0,Y 573.279,Z 386.569,A -85,B 0,C 180,E1 -2036.519,E2 -2036.519} C_VEL
LIN {X 0,Y 573.233,Z 386.579,A -85,B 0,C 180,E1 -2039.116,E2 -2039.116} C_VEL
LIN {X 0,Y 573.26,Z 386.574,A -85,B 0,C 180,E1 -2041.969,E2 -2041.969} C_VEL
LIN {X 0,Y 573.252,Z 386.573,A -85,B 0,C 180,E1 -2044.59,E2 -2044.59} C_VEL
LIN {X 0,Y 573.233,Z 386.58,A -85,B 0,C 180,E1 -2047.663,E2 -2047.663} C_VEL
LIN {X 0,Y 573.274,Z 386.572,A -85,B 0,C 180,E1 -2050.728,E2 -2050.728} C_VEL
LIN {X 0,Y 573.247,Z 386.578,A -85,B 0,C 180,E1 -2053.622,E2 -2053.622} C_VEL
LIN {X 0,Y 573.27,Z 386.573,A -85,B 0,C 180,E1 -2055.807,E2 -2055.807} C_VEL
LIN {X 0,Y 573.259,Z 386.575,A -85,B 0,C 180,E1 -2058.745,E2 -2058.745} C_VEL
LIN {X 0,Y 573.287,Z 386.573,A -85,B 0,C 180,E1 -2061.541,E2 -2061.541} C_VEL
LIN {X 0,Y 573.298,Z 386.569,A -85,B 0,C 180,E1 -2064.372,E2 -2064.372} C_VEL
LIN {X 0,Y 573.314,Z 386.566,A -85,B 0,C 180,E1 -2067.893,E2 -2067.893} C_VEL
LIN {X 0,Y 573.329,Z 386.569,A -85,B 0,C 180,E1 -2070.703,E2 -2070.703} C_VEL
LIN {X 0,Y 573.302,Z 386.575,A -85,B 0,C 180,E1 -2072.811,E2 -2072.811} C_VEL
LIN {X 0,Y 573.298,Z 386.569,A -85,B 0,C 180,E1 -2075.628,E2 -2075.628} C_VEL
LIN {X 0,Y 573.287,Z 386.573,A -85,B 0,C 180,E1 -2078.459,E2 -2078.459} C_VEL
LIN {X 0,Y 573.269,Z 386.574,A -85,B 0,C 180,E1 -2081.312,E2 -2081.312} C_VEL
LIN {X 0,Y 573.27,Z 386.573,A -85,B 0,C 180,E1 -2084.193,E2 -2084.193} C_VEL
LIN {X 0,Y 573.255,Z 386.577,A -85,B 0,C 180,E1 -2087.112,E2 -2087.112} C_VEL
LIN {X 0,Y 573.25,Z 386.574,A -85,B 0,C 180,E1 -2090.077,E2 -2090.077} C_VEL
LIN {X 0,Y 573.23,Z 386.578,A -85,B 0,C 180,E1 -2093.099,E2 -2093.099} C_VEL
LIN {X 0,Y 573.253,Z 386.573,A -85,B 0,C 180,E1 -2095.41,E2 -2095.41} C_VEL
LIN {X 0,Y 573.261,Z 386.574,A -85,B 0,C 180,E1 -2098.032,E2 -2098.032} C_VEL
LIN {X 0,Y 573.234,Z 386.579,A -85,B 0,C 180,E1 -2100.884,E2 -2100.884} C_VEL
LIN {X 0,Y 573.257,Z 386.572,A -85,B 0,C 180,E1 -2103.524,E2 -2103.524} C_VEL
LIN {X 0,Y 573.256,Z 386.576,A -85,B 0,C 180,E1 -2106.048,E2 -2106.048} C_VEL
LIN {X 0,Y 573.244,Z 386.579,A -85,B 0,C 180,E1 -2108.701,E2 -2108.701} C_VEL
LIN {X 0,Y 573.249,Z 386.573,A -85,B 0,C 180,E1 -2111.596,E2 -2111.596} C_VEL
LIN {X 0,Y 573.234,Z 386.585,A -85,B 0,C 180,E1 -2114.333,E2 -2114.333} C_VEL
LIN {X 0,Y 573.235,Z 386.575,A -85,B 0,C 180,E1 -2117.358,E2 -2117.358} C_VEL
LIN {X 0,Y 573.244,Z 386.581,A -85,B 0,C 180,E1 -2120.393,E2 -2120.393} C_VEL
LIN {X 0,Y 573.251,Z 386.573,A -85,B 0,C 180,E1 -2123.078,E2 -2123.078} C_VEL
LIN {X 0,Y 573.269,Z 386.573,A -85,B 0,C 180,E1 -2125.672,E2 -2125.672} C_VEL
LIN {X 0,Y 573.244,Z 386.582,A -85,B 0,C 180,E1 -2128.185,E2 -2128.185} C_VEL
LIN {X 0,Y 573.264,Z 386.573,A -85,B 0,C 180,E1 -2130.635,E2 -2130.635} C_VEL
LIN {X 0,Y 573.25,Z 386.573,A -85,B 0,C 180,E1 -2133.025,E2 -2133.025} C_VEL
LIN {X 0,Y 573.27,Z 386.572,A -85,B 0,C 180,E1 -2135.366,E2 -2135.366} C_VEL
LIN {X 0,Y 573.224,Z 386.579,A -85,B 0,C 180,E1 -2138.42,E2 -2138.42} C_VEL
LIN {X 0,Y 573.273,Z 386.57,A -85,B 0,C 180,E1 -2140.728,E2 -2140.728} C_VEL
LIN {X 0,Y 573.255,Z 386.578,A -85,B 0,C 180,E1 -2143.622,E2 -2143.622} C_VEL
LIN {X 0,Y 573.234,Z 386.576,A -85,B 0,C 180,E1 -2146.53,E2 -2146.53} C_VEL
LIN {X 0,Y 573.257,Z 386.572,A -85,B 0,C 180,E1 -2148.745,E2 -2148.745} C_VEL
LIN {X 0,Y 573.286,Z 386.575,A -85,B 0,C 180,E1 -2151.541,E2 -2151.541} C_VEL
LIN {X 0,Y 573.289,Z 386.569,A -85,B 0,C 180,E1 -2154.372,E2 -2154.372} C_VEL
LIN {X 0,Y 573.305,Z 386.572,A -85,B 0,C 180,E1 -2157.893,E2 -2157.893} C_VEL
LIN {X 0,Y 573.33,Z 386.563,A -85,B 0,C 180,E1 -2160.703,E2 -2160.703} C_VEL
LIN {X 0,Y 573.235,Z 386.584,A -85,B 0,C 180,E1 -2163.515,E2 -2163.515} C_VEL
LIN {X 0,Y 573.289,Z 386.576,A -85,B 0,C 180,E1 -2165.629,E2 -2165.629} C_VEL
LIN {X 0,Y 573.287,Z 386.568,A -85,B 0,C 180,E1 -2168.46,E2 -2168.46} C_VEL
LIN {X 0,Y 573.268,Z 386.579,A -85,B 0,C 180,E1 -2171.312,E2 -2171.312} C_VEL
LIN {X 0,Y 573.27,Z 386.571,A -85,B 0,C 180,E1 -2174.193,E2 -2174.193} C_VEL
LIN {X 0,Y 573.256,Z 386.578,A -85,B 0,C 180,E1 -2177.112,E2 -2177.112} C_VEL
LIN {X 0,Y 573.25,Z 386.573,A -85,B 0,C 180,E1 -2180.077,E2 -2180.077} C_VEL
LIN {X 0,Y 573.231,Z 386.582,A -85,B 0,C 180,E1 -2183.1,E2 -2183.1} C_VEL
LIN {X 0,Y 573.253,Z 386.579,A -85,B 0,C 180,E1 -2185.411,E2 -2185.411} C_VEL
LIN {X 0,Y 573.251,Z 386.573,A -85,B 0,C 180,E1 -2188.03,E2 -2188.03} C_VEL
LIN {X 0,Y 573.238,Z 386.58,A -85,B 0,C 180,E1 -2190.885,E2 -2190.885} C_VEL
LIN {X 0,Y 573.261,Z 386.575,A -85,B 0,C 180,E1 -2193.525,E2 -2193.525} C_VEL
LIN {X 0,Y 573.26,Z 386.572,A -85,B 0,C 180,E1 -2196.049,E2 -2196.049} C_VEL
LIN {X 0,Y 573.249,Z 386.579,A -85,B 0,C 180,E1 -2198.701,E2 -2198.701} C_VEL
LIN {X 0,Y 573.253,Z 386.576,A -85,B 0,C 180,E1 -2201.596,E2 -2201.596} C_VEL
LIN {X 0,Y 573.235,Z 386.579,A -85,B 0,C 180,E1 -2204.334,E2 -2204.334} C_VEL
LIN {X 0,Y 573.248,Z 386.582,A -85,B 0,C 180,E1 -2206.642,E2 -2206.642} C_VEL
LIN {X 0,Y 573.391,Z 387.538,A -85,B 0,C 180,E1 -2207.614,E2 -2207.614} C_VEL
LIN {X 0,Y 573.578,Z 390.676,A -85,B 0,C 180,E1 -2209.504,E2 -2209.504} C_VEL
LIN {X 0,Y 573.416,Z 395.573,A -85,B 0,C 180,E1 -2212.207,E2 -2212.207} C_VEL
LIN {X 0,Y 573.327,Z 400.751,A -85,B 0,C 180,E1 -2214.821,E2 -2214.821} C_VEL
LIN {X 0,Y 573.292,Z 406.141,A -85,B 0,C 180,E1 -2217.358,E2 -2217.358} C_VEL
LIN {X 0,Y 573.247,Z 411.53,A -85,B 0,C 180,E1 -2219.824,E2 -2219.824} C_VEL
LIN {X 0,Y 573.19,Z 416.92,A -85,B 0,C 180,E1 -2222.23,E2 -2222.23} C_VEL
LIN {X 0,Y 573.175,Z 423.597,A -85,B 0,C 180,E1 -2225.143,E2 -2225.143} C_VEL
LIN {X 0,Y 573.118,Z 429.495,A -85,B 0,C 180,E1 -2227.658,E2 -2227.658} C_VEL
LIN {X 0,Y 573.08,Z 434.885,A -85,B 0,C 180,E1 -2229.917,E2 -2229.917} C_VEL
LIN {X 0,Y 573.082,Z 440.274,A -85,B 0,C 180,E1 -2232.146,E2 -2232.146} C_VEL
LIN {X 0,Y 573.048,Z 447.46,A -85,B 0,C 180,E1 -2235.075,E2 -2235.075} C_VEL
LIN {X 0,Y 573.004,Z 453.523,A -85,B 0,C 180,E1 -2237.516,E2 -2237.516} C_VEL
LIN {X 0,Y 573.856,Z 459.527,A -85,B 0,C 180,E1 -2237.647,E2 -2237.647} C_VEL
LIN {X 0,Y 573.782,Z 471.835,A -85,B 0,C 180,E1 -2237.982,E2 -2237.982} C_VEL
LIN {X 0,Y 573.67,Z 482.271,A -85,B 0,C 180,E1 -2238.374,E2 -2238.374} C_VEL
LIN {X 0,Y 573.551,Z 494.269,A -85,B 0,C 180,E1 -2238.966,E2 -2238.966} C_VEL
LIN {X 0,Y 573.453,Z 505.48,A -85,B 0,C 180,E1 -2239.675,E2 -2239.675} C_VEL
LIN {X 0,Y 573.307,Z 515.642,A -85,B 0,C 180,E1 -2240.474,E2 -2240.474} C_VEL
LIN {X 0,Y 573.214,Z 524.767,A -85,B 0,C 180,E1 -2241.362,E2 -2241.362} C_VEL
LIN {X 0,Y 573.16,Z 532.316,A -85,B 0,C 180,E1 -2242.248,E2 -2242.248} C_VEL
LIN {X 0,Y 573.065,Z 539.701,A -85,B 0,C 180,E1 -2243.304,E2 -2243.304} C_VEL
LIN {X 0,Y 573.068,Z 545.681,A -85,B 0,C 180,E1 -2244.37,E2 -2244.37} C_VEL
LIN {X 0,Y 573.028,Z 550.376,A -85,B 0,C 180,E1 -2245.427,E2 -2245.427} C_VEL
LIN {X 0,Y 573.022,Z 553.962,A -85,B 0,C 180,E1 -2246.484,E2 -2246.484} C_VEL
LIN {X 0,Y 572.959,Z 555.797,A -85,B 0,C 180,E1 -2247.188,E2 -2247.188} C_VEL
LIN {X 0,Y 572.946,Z 558.188,A -85,B 0,C 180,E1 -2248.594,E2 -2248.594} C_VEL
LIN {X 0,Y 572.941,Z 558.782,A -85,B 0,C 180,E1 -2249.297,E2 -2249.297} C_VEL
LIN {X 0,Y 572.938,Z 558.979,A -85,B 0,C 180,E1 -2250,E2 -2250} C_VEL
LIN {X 0,Y 572.941,Z 558.782,A -85,B 0,C 180,E1 -2250.703,E2 -2250.703} C_VEL
LIN {X 0,Y 572.946,Z 558.188,A -85,B 0,C 180,E1 -2251.406,E2 -2251.406} C_VEL
LIN {X 0,Y 572.959,Z 555.798,A -85,B 0,C 180,E1 -2252.812,E2 -2252.812} C_VEL
LIN {X 0,Y 573.014,Z 552.887,A -85,B 0,C 180,E1 -2253.868,E2 -2253.868} C_VEL
LIN {X 0,Y 572.962,Z 548.939,A -85,B 0,C 180,E1 -2254.925,E2 -2254.925} C_VEL
LIN {X 0,Y 573.073,Z 543.845,A -85,B 0,C 180,E1 -2255.983,E2 -2255.983} C_VEL
LIN {X 0,Y 573.082,Z 537.462,A -85,B 0,C 180,E1 -2257.044,E2 -2257.044} C_VEL
LIN {X 0,Y 573.177,Z 529.489,A -85,B 0,C 180,E1 -2258.106,E2 -2258.106} C_VEL
LIN {X 0,Y 573.279,Z 521.348,A -85,B 0,C 180,E1 -2258.992,E2 -2258.992} C_VEL
LIN {X 0,Y 573.349,Z 511.372,A -85,B 0,C 180,E1 -2259.881,E2 -2259.881} C_VEL
LIN {X 0,Y 573.491,Z 501.556,A -85,B 0,C 180,E1 -2260.592,E2 -2260.592} C_VEL
LIN {X 0,Y 573.598,Z 490.319,A -85,B 0,C 180,E1 -2261.247,E2 -2261.247} C_VEL
LIN {X 0,Y 573.704,Z 476.999,A -85,B 0,C 180,E1 -2261.84,E2 -2261.84} C_VEL
LIN {X 0,Y 573.836,Z 464.145,A -85,B 0,C 180,E1 -2262.241,E2 -2262.241} C_VEL
LIN {X 0,Y 573.672,Z 457.558,A -85,B 0,C 180,E1 -2262.396,E2 -2262.396} C_VEL
LIN {X 0,Y 573.004,Z 453.532,A -85,B 0,C 180,E1 -2262.484,E2 -2262.484} C_VEL
LIN {X 0,Y 573.048,Z 447.461,A -85,B 0,C 180,E1 -2264.924,E2 -2264.924} C_VEL
LIN {X 0,Y 573.081,Z 440.275,A -85,B 0,C 180,E1 -2267.853,E2 -2267.853} C_VEL
LIN {X 0,Y 573.079,Z 434.885,A -85,B 0,C 180,E1 -2270.082,E2 -2270.082} C_VEL
LIN {X 0,Y 573.118,Z 429.496,A -85,B 0,C 180,E1 -2272.342,E2 -2272.342} C_VEL
LIN {X 0,Y 573.153,Z 422.31,A -85,B 0,C 180,E1 -2275.414,E2 -2275.414} C_VEL
LIN {X 0,Y 573.203,Z 416.355,A -85,B 0,C 180,E1 -2278.019,E2 -2278.019} C_VEL
LIN {X 0,Y 573.25,Z 411.531,A -85,B 0,C 180,E1 -2280.175,E2 -2280.175} C_VEL
LIN {X 0,Y 573.291,Z 406.141,A -85,B 0,C 180,E1 -2282.642,E2 -2282.642} C_VEL
LIN {X 0,Y 573.326,Z 400.752,A -85,B 0,C 180,E1 -2285.179,E2 -2285.179} C_VEL
LIN {X 0,Y 573.414,Z 395.573,A -85,B 0,C 180,E1 -2287.793,E2 -2287.793} C_VEL
LIN {X 0,Y 573.583,Z 390.556,A -85,B 0,C 180,E1 -2290.564,E2 -2290.564} C_VEL
LIN {X 0,Y 573.333,Z 387.117,A -85,B 0,C 180,E1 -2292.651,E2 -2292.651} C_VEL
LIN {X 0,Y 573.251,Z 386.579,A -85,B 0,C 180,E1 -2293.669,E2 -2293.669} C_VEL
LIN {X 0,Y 573.237,Z 386.58,A -85,B 0,C 180,E1 -2296.64,E2 -2296.64} C_VEL
LIN {X 0,Y 573.271,Z 386.575,A -85,B 0,C 180,E1 -2299.477,E2 -2299.477} C_VEL
LIN {X 0,Y 573.234,Z 386.576,A -85,B 0,C 180,E1 -2302.192,E2 -2302.192} C_VEL
LIN {X 0,Y 573.265,Z 386.58,A -85,B 0,C 180,E1 -2304.816,E2 -2304.816} C_VEL
LIN {X 0,Y 573.251,Z 386.576,A -85,B 0,C 180,E1 -2307.354,E2 -2307.354} C_VEL
LIN {X 0,Y 573.253,Z 386.572,A -85,B 0,C 180,E1 -2309.824,E2 -2309.824} C_VEL
LIN {X 0,Y 573.285,Z 386.57,A -85,B 0,C 180,E1 -2312.234,E2 -2312.234} C_VEL
LIN {X 0,Y 573.271,Z 386.572,A -85,B 0,C 180,E1 -2315.366,E2 -2315.366} C_VEL
LIN {X 0,Y 573.225,Z 386.581,A -85,B 0,C 180,E1 -2318.419,E2 -2318.419} C_VEL
LIN {X 0,Y 573.272,Z 386.58,A -85,B 0,C 180,E1 -2320.728,E2 -2320.728} C_VEL
LIN {X 0,Y 573.254,Z 386.572,A -85,B 0,C 180,E1 -2323.621,E2 -2323.621} C_VEL
LIN {X 0,Y 573.234,Z 386.584,A -85,B 0,C 180,E1 -2326.529,E2 -2326.529} C_VEL
LIN {X 0,Y 573.256,Z 386.579,A -85,B 0,C 180,E1 -2328.744,E2 -2328.744} C_VEL
LIN {X 0,Y 573.285,Z 386.568,A -85,B 0,C 180,E1 -2331.54,E2 -2331.54} C_VEL
LIN {X 0,Y 573.288,Z 386.576,A -85,B 0,C 180,E1 -2334.371,E2 -2334.371} C_VEL
LIN {X 0,Y 573.304,Z 386.568,A -85,B 0,C 180,E1 -2337.892,E2 -2337.892} C_VEL
LIN {X 0,Y 573.329,Z 386.568,A -85,B 0,C 180,E1 -2340.702,E2 -2340.702} C_VEL
LIN {X 0,Y 573.234,Z 386.575,A -85,B 0,C 180,E1 -2343.514,E2 -2343.514} C_VEL
LIN {X 0,Y 573.288,Z 386.569,A -85,B 0,C 180,E1 -2345.628,E2 -2345.628} C_VEL
LIN {X 0,Y 573.285,Z 386.575,A -85,B 0,C 180,E1 -2348.459,E2 -2348.459} C_VEL
LIN {X 0,Y 573.263,Z 386.571,A -85,B 0,C 180,E1 -2351.312,E2 -2351.312} C_VEL
LIN {X 0,Y 573.267,Z 386.581,A -85,B 0,C 180,E1 -2354.193,E2 -2354.193} C_VEL
LIN {X 0,Y 573.253,Z 386.572,A -85,B 0,C 180,E1 -2357.111,E2 -2357.111} C_VEL
LIN {X 0,Y 573.247,Z 386.583,A -85,B 0,C 180,E1 -2360.076,E2 -2360.076} C_VEL
LIN {X 0,Y 573.226,Z 386.576,A -85,B 0,C 180,E1 -2363.099,E2 -2363.099} C_VEL
LIN {X 0,Y 573.244,Z 386.575,A -85,B 0,C 180,E1 -2364.394,E2 -2364.394} C_VEL
LIN {X 0,Y 572.618,Z 386.655,A -85,B 0,C 180,E1 -2364.981,E2 -2364.981} C_VEL
LIN {X 0,Y 569.781,Z 387.014,A -85,B 0,C 180,E1 -2365.933,E2 -2365.933} C_VEL
LIN {X 0,Y 567.353,Z 387.312,A -85,B 0,C 180,E1 -2366.698,E2 -2366.698} C_VEL
LIN {X 0,Y 566.3,Z 387.44,A -85,B 0,C 180,E1 -2367.29,E2 -2367.29} C_VEL
LIN {X 0,Y 566.211,Z 387.451,A -85,B 0,C 180,E1 -2367.49,E2 -2367.49} C_VEL
LIN {X 0,Y 566.187,Z 387.454,A -85,B 0,C 180,E1 -2370.592,E2 -2370.592} C_VEL
LIN {X 0,Y 566.221,Z 387.449,A -85,B 0,C 180,E1 -2373.102,E2 -2373.102} C_VEL
LIN {X 0,Y 566.205,Z 387.458,A -85,B 0,C 180,E1 -2375.688,E2 -2375.688} C_VEL
LIN {X 0,Y 566.21,Z 387.45,A -85,B 0,C 180,E1 -2378.559,E2 -2378.559} C_VEL
LIN {X 0,Y 566.205,Z 387.452,A -85,B 0,C 180,E1 -2381.136,E2 -2381.136} C_VEL
LIN {X 0,Y 566.193,Z 387.457,A -85,B 0,C 180,E1 -2384.036,E2 -2384.036} C_VEL
LIN {X 0,Y 566.203,Z 387.452,A -85,B 0,C 180,E1 -2387.082,E2 -2387.082} C_VEL
LIN {X 0,Y 566.22,Z 387.455,A -85,B 0,C 180,E1 -2389.803,E2 -2389.803} C_VEL
LIN {X 0,Y 566.193,Z 387.452,A -85,B 0,C 180,E1 -2392.599,E2 -2392.599} C_VEL
LIN {X 0,Y 566.214,Z 387.454,A -85,B 0,C 180,E1 -2395.183,E2 -2395.183} C_VEL
LIN {X 0,Y 566.231,Z 387.453,A -85,B 0,C 180,E1 -2397.744,E2 -2397.744} C_VEL
LIN {X 0,Y 566.198,Z 387.451,A -85,B 0,C 180,E1 -2400.328,E2 -2400.328} C_VEL
LIN {X 0,Y 566.22,Z 387.449,A -85,B 0,C 180,E1 -2402.662,E2 -2402.662} C_VEL
LIN {X 0,Y 566.231,Z 387.451,A -85,B 0,C 180,E1 -2405.039,E2 -2405.039} C_VEL
LIN {X 0,Y 566.19,Z 387.453,A -85,B 0,C 180,E1 -2408.138,E2 -2408.138} C_VEL
LIN {X 0,Y 566.232,Z 387.448,A -85,B 0,C 180,E1 -2410.612,E2 -2410.612} C_VEL
LIN {X 0,Y 566.211,Z 387.458,A -85,B 0,C 180,E1 -2413.413,E2 -2413.413} C_VEL
LIN {X 0,Y 566.195,Z 387.453,A -85,B 0,C 180,E1 -2416.359,E2 -2416.359} C_VEL
LIN {X 0,Y 566.231,Z 387.45,A -85,B 0,C 180,E1 -2418.675,E2 -2418.675} C_VEL
LIN {X 0,Y 566.23,Z 387.453,A -85,B 0,C 180,E1 -2421.435,E2 -2421.435} C_VEL
LIN {X 0,Y 566.267,Z 387.444,A -85,B 0,C 180,E1 -2424.302,E2 -2424.302} C_VEL
LIN {X 0,Y 566.284,Z 387.442,A -85,B 0,C 180,E1 -2427.866,E2 -2427.866} C_VEL
LIN {X 0,Y 566.3,Z 387.445,A -85,B 0,C 180,E1 -2430.711,E2 -2430.711} C_VEL
LIN {X 0,Y 566.269,Z 387.452,A -85,B 0,C 180,E1 -2432.846,E2 -2432.846} C_VEL
LIN {X 0,Y 566.267,Z 387.444,A -85,B 0,C 180,E1 -2435.698,E2 -2435.698} C_VEL
LIN {X 0,Y 566.231,Z 387.453,A -85,B 0,C 180,E1 -2438.566,E2 -2438.566} C_VEL
LIN {X 0,Y 566.239,Z 387.448,A -85,B 0,C 180,E1 -2441.454,E2 -2441.454} C_VEL
LIN {X 0,Y 566.231,Z 387.454,A -85,B 0,C 180,E1 -2444.507,E2 -2444.507} C_VEL
LIN {X 0,Y 566.197,Z 387.454,A -85,B 0,C 180,E1 -2447.332,E2 -2447.332} C_VEL
LIN {X 0,Y 566.211,Z 387.454,A -85,B 0,C 180,E1 -2450.337,E2 -2450.337} C_VEL
LIN {X 0,Y 566.186,Z 387.453,A -85,B 0,C 180,E1 -2453.404,E2 -2453.404} C_VEL
LIN {X 0,Y 566.222,Z 387.448,A -85,B 0,C 180,E1 -2455.748,E2 -2455.748} C_VEL
LIN {X 0,Y 566.203,Z 387.455,A -85,B 0,C 180,E1 -2458.203,E2 -2458.203} C_VEL
LIN {X 0,Y 566.195,Z 387.454,A -85,B 0,C 180,E1 -2461.078,E2 -2461.078} C_VEL
LIN {X 0,Y 566.208,Z 387.451,A -85,B 0,C 180,E1 -2463.734,E2 -2463.734} C_VEL
LIN {X 0,Y 566.212,Z 387.457,A -85,B 0,C 180,E1 -2466.569,E2 -2466.569} C_VEL
LIN {X 0,Y 566.207,Z 387.451,A -85,B 0,C 180,E1 -2469.686,E2 -2469.686} C_VEL
LIN {X 0,Y 566.212,Z 387.455,A -85,B 0,C 180,E1 -2472.087,E2 -2472.087} C_VEL
LIN {X 0,Y 566.168,Z 387.456,A -85,B 0,C 180,E1 -2475.036,E2 -2475.036} C_VEL
LIN {X 0,Y 566.213,Z 387.457,A -85,B 0,C 180,E1 -2478.136,E2 -2478.136} C_VEL
LIN {X 0,Y 566.218,Z 387.451,A -85,B 0,C 180,E1 -2480.727,E2 -2480.727} C_VEL
LIN {X 0,Y 566.213,Z 387.453,A -85,B 0,C 180,E1 -2483.783,E2 -2483.783} C_VEL
LIN {X 0,Y 566.207,Z 387.458,A -85,B 0,C 180,E1 -2486.266,E2 -2486.266} C_VEL
LIN {X 0,Y 566.197,Z 387.452,A -85,B 0,C 180,E1 -2488.922,E2 -2488.922} C_VEL
LIN {X 0,Y 566.19,Z 387.452,A -85,B 0,C 180,E1 -2491.047,E2 -2491.047} C_VEL
LIN {X 0,Y 566.214,Z 387.451,A -85,B 0,C 180,E1 -2493.459,E2 -2493.459} C_VEL
LIN {X 0,Y 566.195,Z 387.459,A -85,B 0,C 180,E1 -2495.82,E2 -2495.82} C_VEL
LIN {X 0,Y 566.203,Z 387.451,A -85,B 0,C 180,E1 -2498.903,E2 -2498.903} C_VEL
LIN {X 0,Y 566.207,Z 387.451,A -85,B 0,C 180,E1 -2501.173,E2 -2501.173} C_VEL
LIN {X 0,Y 566.216,Z 387.452,A -85,B 0,C 180,E1 -2503.413,E2 -2503.413} C_VEL
LIN {X 0,Y 566.196,Z 387.454,A -85,B 0,C 180,E1 -2506.359,E2 -2506.359} C_VEL
LIN {X 0,Y 566.229,Z 387.447,A -85,B 0,C 180,E1 -2508.675,E2 -2508.675} C_VEL
LIN {X 0,Y 566.23,Z 387.452,A -85,B 0,C 180,E1 -2511.435,E2 -2511.435} C_VEL
LIN {X 0,Y 566.257,Z 387.445,A -85,B 0,C 180,E1 -2514.302,E2 -2514.302} C_VEL
LIN {X 0,Y 566.276,Z 387.448,A -85,B 0,C 180,E1 -2517.867,E2 -2517.867} C_VEL
LIN {X 0,Y 566.3,Z 387.439,A -85,B 0,C 180,E1 -2520.711,E2 -2520.711} C_VEL
LIN {X 0,Y 566.272,Z 387.443,A -85,B 0,C 180,E1 -2522.846,E2 -2522.846} C_VEL
LIN {X 0,Y 566.257,Z 387.451,A -85,B 0,C 180,E1 -2525.699,E2 -2525.699} C_VEL
LIN {X 0,Y 566.231,Z 387.447,A -85,B 0,C 180,E1 -2528.566,E2 -2528.566} C_VEL
LIN {X 0,Y 566.238,Z 387.456,A -85,B 0,C 180,E1 -2531.455,E2 -2531.455} C_VEL
LIN {X 0,Y 566.231,Z 387.447,A -85,B 0,C 180,E1 -2534.507,E2 -2534.507} C_VEL
LIN {X 0,Y 566.201,Z 387.461,A -85,B 0,C 180,E1 -2537.332,E2 -2537.332} C_VEL
LIN {X 0,Y 566.211,Z 387.449,A -85,B 0,C 180,E1 -2540.338,E2 -2540.338} C_VEL
LIN {X 0,Y 566.187,Z 387.46,A -85,B 0,C 180,E1 -2543.404,E2 -2543.404} C_VEL
LIN {X 0,Y 566.212,Z 387.452,A -85,B 0,C 180,E1 -2545.749,E2 -2545.749} C_VEL
LIN {X 0,Y 566.2,Z 387.451,A -85,B 0,C 180,E1 -2548.203,E2 -2548.203} C_VEL
LIN {X 0,Y 566.198,Z 387.46,A -85,B 0,C 180,E1 -2551.079,E2 -2551.079} C_VEL
LIN {X 0,Y 566.211,Z 387.451,A -85,B 0,C 180,E1 -2553.735,E2 -2553.735} C_VEL
LIN {X 0,Y 566.216,Z 387.453,A -85,B 0,C 180,E1 -2556.569,E2 -2556.569} C_VEL
LIN {X 0,Y 566.213,Z 387.452,A -85,B 0,C 180,E1 -2559.686,E2 -2559.686} C_VEL
LIN {X 0,Y 566.213,Z 387.452,A -85,B 0,C 180,E1 -2562.088,E2 -2562.088} C_VEL
LIN {X 0,Y 566.174,Z 387.463,A -85,B 0,C 180,E1 -2565.036,E2 -2565.036} C_VEL
LIN {X 0,Y 566.203,Z 387.457,A -85,B 0,C 180,E1 -2566.049,E2 -2566.049} C_VEL
LIN {X 0,Y 566.298,Z 388.014,A -85,B 0,C 180,E1 -2567.073,E2 -2567.073} C_VEL
LIN {X 0,Y 566.59,Z 391.379,A -85,B 0,C 180,E1 -2569.17,E2 -2569.17} C_VEL
LIN {X 0,Y 566.482,Z 395.82,A -85,B 0,C 180,E1 -2571.661,E2 -2571.661} C_VEL
LIN {X 0,Y 566.323,Z 400.761,A -85,B 0,C 180,E1 -2574.32,E2 -2574.32} C_VEL
LIN {X 0,Y 566.286,Z 406.141,A -85,B 0,C 180,E1 -2576.903,E2 -2576.903} C_VEL
LIN {X 0,Y 566.197,Z 411.53,A -85,B 0,C 180,E1 -2579.409,E2 -2579.409} C_VEL
LIN {X 0,Y 566.15,Z 416.92,A -85,B 0,C 180,E1 -2581.854,E2 -2581.854} C_VEL
LIN {X 0,Y 566.11,Z 422.309,A -85,B 0,C 180,E1 -2584.246,E2 -2584.246} C_VEL
LIN {X 0,Y 566.073,Z 428.05,A -85,B 0,C 180,E1 -2586.743,E2 -2586.743} C_VEL
LIN {X 0,Y 566.018,Z 434.885,A -85,B 0,C 180,E1 -2589.656,E2 -2589.656} C_VEL
LIN {X 0,Y 566.003,Z 440.274,A -85,B 0,C 180,E1 -2591.915,E2 -2591.915} C_VEL
LIN {X 0,Y 565.957,Z 447.46,A -85,B 0,C 180,E1 -2594.884,E2 -2594.884} C_VEL
LIN {X 0,Y 565.914,Z 453.523,A -85,B 0,C 180,E1 -2597.357,E2 -2597.357} C_VEL
LIN {X 0,Y 566.923,Z 460.496,A -85,B 0,C 180,E1 -2597.516,E2 -2597.516} C_VEL
LIN {X 0,Y 566.822,Z 473.123,A -85,B 0,C 180,E1 -2597.877,E2 -2597.877} C_VEL
LIN {X 0,Y 566.704,Z 483.477,A -85,B 0,C 180,E1 -2598.284,E2 -2598.284} C_VEL
LIN {X 0,Y 566.576,Z 494.701,A -85,B 0,C 180,E1 -2598.853,E2 -2598.853} C_VEL
LIN {X 0,Y 566.445,Z 506.748,A -85,B 0,C 180,E1 -2599.636,E2 -2599.636} C_VEL
LIN {X 0,Y 566.301,Z 515.64,A -85,B 0,C 180,E1 -2600.355,E2 -2600.355} C_VEL
LIN {X 0,Y 566.166,Z 524.764,A -85,B 0,C 180,E1 -2601.253,E2 -2601.253} C_VEL
LIN {X 0,Y 566.094,Z 532.312,A -85,B 0,C 180,E1 -2602.151,E2 -2602.151} C_VEL
LIN {X 0,Y 565.998,Z 539.956,A -85,B 0,C 180,E1 -2603.261,E2 -2603.261} C_VEL
LIN {X 0,Y 565.998,Z 545.681,A -85,B 0,C 180,E1 -2604.299,E2 -2604.299} C_VEL
LIN {X 0,Y 565.933,Z 550.377,A -85,B 0,C 180,E1 -2605.37,E2 -2605.37} C_VEL
LIN {X 0,Y 565.927,Z 553.964,A -85,B 0,C 180,E1 -2606.44,E2 -2606.44} C_VEL
LIN {X 0,Y 565.878,Z 555.795,A -85,B 0,C 180,E1 -2607.152,E2 -2607.152} C_VEL
LIN {X 0,Y 565.846,Z 558.189,A -85,B 0,C 180,E1 -2608.576,E2 -2608.576} C_VEL
LIN {X 0,Y 565.841,Z 558.782,A -85,B 0,C 180,E1 -2609.288,E2 -2609.288} C_VEL
LIN {X 0,Y 565.841,Z 558.782,A -85,B 0,C 180,E1 -2610.711,E2 -2610.711} C_VEL
LIN {X 0,Y 565.846,Z 558.189,A -85,B 0,C 180,E1 -2611.423,E2 -2611.423} C_VEL
LIN {X 0,Y 565.878,Z 555.795,A -85,B 0,C 180,E1 -2612.847,E2 -2612.847} C_VEL
LIN {X 0,Y 565.926,Z 552.884,A -85,B 0,C 180,E1 -2613.916,E2 -2613.916} C_VEL
LIN {X 0,Y 565.878,Z 548.935,A -85,B 0,C 180,E1 -2614.987,E2 -2614.987} C_VEL
LIN {X 0,Y 565.99,Z 543.84,A -85,B 0,C 180,E1 -2616.058,E2 -2616.058} C_VEL
LIN {X 0,Y 566.032,Z 537.457,A -85,B 0,C 180,E1 -2617.132,E2 -2617.132} C_VEL
LIN {X 0,Y 566.133,Z 529.49,A -85,B 0,C 180,E1 -2618.207,E2 -2618.207} C_VEL
LIN {X 0,Y 566.238,Z 521.349,A -85,B 0,C 180,E1 -2619.105,E2 -2619.105} C_VEL
LIN {X 0,Y 566.35,Z 511.366,A -85,B 0,C 180,E1 -2620.004,E2 -2620.004} C_VEL
LIN {X 0,Y 566.508,Z 501.549,A -85,B 0,C 180,E1 -2620.724,E2 -2620.724} C_VEL
LIN {X 0,Y 566.603,Z 490.321,A -85,B 0,C 180,E1 -2621.388,E2 -2621.388} C_VEL
LIN {X 0,Y 566.752,Z 476.994,A -85,B 0,C 180,E1 -2621.988,E2 -2621.988} C_VEL
LIN {X 0,Y 566.896,Z 464.129,A -85,B 0,C 180,E1 -2622.393,E2 -2622.393} C_VEL
LIN {X 0,Y 566.636,Z 457.847,A -85,B 0,C 180,E1 -2622.547,E2 -2622.547} C_VEL
LIN {X 0,Y 565.914,Z 453.524,A -85,B 0,C 180,E1 -2622.643,E2 -2622.643} C_VEL
LIN {X 0,Y 565.957,Z 447.461,A -85,B 0,C 180,E1 -2625.116,E2 -2625.116} C_VEL
LIN {X 0,Y 566.003,Z 440.275,A -85,B 0,C 180,E1 -2628.084,E2 -2628.084} C_VEL
LIN {X 0,Y 566.018,Z 434.885,A -85,B 0,C 180,E1 -2630.344,E2 -2630.344} C_VEL
LIN {X 0,Y 566.072,Z 428.05,A -85,B 0,C 180,E1 -2633.257,E2 -2633.257} C_VEL
LIN {X 0,Y 566.109,Z 422.31,A -85,B 0,C 180,E1 -2635.754,E2 -2635.754} C_VEL
LIN {X 0,Y 566.148,Z 416.819,A -85,B 0,C 180,E1 -2638.191,E2 -2638.191} C_VEL
LIN {X 0,Y 566.198,Z 411.531,A -85,B 0,C 180,E1 -2640.591,E2 -2640.591} C_VEL
LIN {X 0,Y 566.284,Z 406.141,A -85,B 0,C 180,E1 -2643.097,E2 -2643.097} C_VEL
LIN {X 0,Y 566.322,Z 400.762,A -85,B 0,C 180,E1 -2645.68,E2 -2645.68} C_VEL
LIN {X 0,Y 566.517,Z 395.345,A -85,B 0,C 180,E1 -2648.596,E2 -2648.596} C_VEL
LIN {X 0,Y 566.585,Z 390.904,A -85,B 0,C 180,E1 -2651.102,E2 -2651.102} C_VEL
LIN {X 0,Y 566.252,Z 387.827,A -85,B 0,C 180,E1 -2653.048,E2 -2653.048} C_VEL
LIN {X 0,Y 566.199,Z 387.457,A -85,B 0,C 180,E1 -2654.035,E2 -2654.035} C_VEL
LIN {X 0,Y 566.2,Z 387.461,A -85,B 0,C 180,E1 -2657.082,E2 -2657.082} C_VEL
LIN {X 0,Y 566.225,Z 387.45,A -85,B 0,C 180,E1 -2659.802,E2 -2659.802} C_VEL
LIN {X 0,Y 566.196,Z 387.457,A -85,B 0,C 180,E1 -2662.598,E2 -2662.598} C_VEL
LIN {X 0,Y 566.218,Z 387.454,A -85,B 0,C 180,E1 -2665.182,E2 -2665.182} C_VEL
LIN {X 0,Y 566.23,Z 387.447,A -85,B 0,C 180,E1 -2667.743,E2 -2667.743} C_VEL
LIN {X 0,Y 566.224,Z 387.45,A -85,B 0,C 180,E1 -2670.323,E2 -2670.323} C_VEL
